(* Logix 5000 project; controller FRCFMS vendor 1 type 14 code 150 rev 33.11; software revision 33.00 *)
// FRCFMS

TASK MainTask (continuous, watchdog 500 ms) : MainProgram, ModbusSlaveTCP

MODULES
   Local : vendor 1 type 14 code 150 (Compact 0, rev 33.11)
      Counters : Embedded (Compact 3, rev 1.1, Output RPI 20 ms)
      Discrete_IO : Embedded (Compact 1, rev 3.1, Output RPI 20 ms)
      Analog_IO : Embedded (Compact 2, rev 1.1, Output RPI 80 ms)
      Blue_Driver_Station : vendor 1 type 7 code 357 (Ethernet 10.0.100.42, rev 1.1, Output RPI 20 ms)
      Red_Driver_Station : vendor 1 type 7 code 357 (Ethernet 10.0.100.41, rev 1.1, Output RPI 20 ms)
      Cargo_Ship : vendor 1 type 7 code 357 (Ethernet 10.0.100.43, rev 1.1, Output RPI 20 ms)
END_MODULES

TYPE AcceptResponse :
STRUCT
   Instance : DINT;
   Addr : SockAddr;
END_STRUCT
END_TYPE

TYPE READ_DATA_REQ :
STRUCT
   Timeout : DINT;
   BufLen : DINT;
END_STRUCT
END_TYPE

TYPE READ_RESP_STR :
STRUCT
   FromAddr : SockAddr;
   Buf : STR_4096;
END_STRUCT
END_TYPE

TYPE REQUEST_PARAMETERS :
STRUCT
   Type : DINT;
   Addr : SockAddr;
END_STRUCT
END_TYPE

TYPE SockAddr :
STRUCT
   Family : INT;
   Port : INT;
   Addr : DINT;
END_STRUCT
END_TYPE

TYPE STR_1 :
STRUCT
   LEN : DINT;
   DATA : SINT[1];
END_STRUCT
END_TYPE

TYPE STR_4096 :
STRUCT
   LEN : DINT;
   DATA : SINT[4096];
END_STRUCT
END_TYPE

TYPE STR_462 :
STRUCT
   LEN : DINT;
   DATA : SINT[462];
END_STRUCT
END_TYPE

TYPE STR_OUT :
STRUCT
   LEN : DINT;
   BUFF : SINT[480];
END_STRUCT
END_TYPE

TYPE WRT_DATA :
STRUCT
   Timeout : DINT;
   ToAddr : SockAddr;
   Buffer : STR_OUT;
END_STRUCT
END_TYPE

VAR_GLOBAL   (* controller tags *)
   AllianceDisconnectedFlasher : TIMER := (PRE := 1000, ACC := 928, EN := 1, TT := 1);
   BlueBypass1 : BOOL;
   BlueBypass2 : BOOL;
   BlueBypass3 : BOOL;
   BlueConnected1 : BOOL;
   BlueConnected2 : BOOL;
   BlueConnected3 : BOOL;
   BlueESTOP1 : ALIAS FOR Blue_Driver_Station:I.Data.1;
   BlueESTOP1Light : ALIAS FOR Blue_Driver_Station:O.Data.15;
   BlueESTOP2 : ALIAS FOR Blue_Driver_Station:I.Data.3;
   BlueESTOP2Light : ALIAS FOR Blue_Driver_Station:O.Data.13;
   BlueESTOP3 : ALIAS FOR Blue_Driver_Station:I.Data.5;
   BlueESTOP3Light : ALIAS FOR Blue_Driver_Station:O.Data.11;
   BlueSoftwareESTOP1 : BOOL;
   BlueSoftwareESTOP2 : BOOL;
   BlueSoftwareESTOP3 : BOOL;
   BlueStackStatus1 : ALIAS FOR Blue_Driver_Station:O.Data.14;
   BlueStackStatus2 : ALIAS FOR Blue_Driver_Station:O.Data.12;
   BlueStackStatus3 : ALIAS FOR Blue_Driver_Station:O.Data.10;
   EStop_Light_flasher : TIMER := (PRE := 750);
   Field_Reset_Green : BOOL;
   FieldESTOP : BOOL;
   FieldESTOPButton : ALIAS FOR Local:1:I.Data.0;
   FieldESTOPLight : ALIAS FOR Local:1:O.Data.0;
   Latch_reset : TIMER := (PRE := 50, ACC := 50, EN := 1, DN := 1);
   LostComm : TIMER := (PRE := 5000, ACC := 5000);
   MatchStart : BOOL;
   MatchStartONS : BOOL;
   MatchSYNC : TIMER := (PRE := 1000);
   MBTI_Buf_Len_Sent : DINT := 11;
   MBTI_Change_Log_MSG : MESSAGE;
        MessageParameters(ServiceCode := 16#0010, LocalElement := MBTU_Log_Enable, ...)
   MBTI_Conn_Acc_Timeout_MSG : MESSAGE;
        MessageParameters(ServiceCode := 16#0010, LocalElement := MBTU_Inactivity_Timeout, ...)
   MBTI_Conn_Accept_MSG : MESSAGE;
        MessageParameters(ServiceCode := 16#0050, LocalElement := MBTU_Sock_Accept_Timeout, DestinationTag := MBTI_Sock_Accept_Resp, ...)
   MBTI_ConnectionsLastErrors : DINT;
   MBTI_Create_Sock_MSG : MESSAGE;
        MessageParameters(ServiceCode := 16#004b, LocalElement := MBTI_Socket_Param, DestinationTag := MBTI_Instance, ...)
   MBTI_Delete_All_MSG : MESSAGE;
        MessageParameters(ServiceCode := 16#0051, ...)
   MBTI_Instance : DINT := 25408;
   MBTI_Read_Data_MSG_00 : MESSAGE;
        MessageParameters(ServiceCode := 16#004d, LocalElement := MBTI_Read_Data_Req[0], DestinationTag := MBTI_Read_Resp[0], ...)
   MBTI_Read_Data_MSG_01 : MESSAGE;
        MessageParameters(ServiceCode := 16#004d, LocalElement := MBTI_Read_Data_Req[0], DestinationTag := MBTI_Read_Resp[1], ...)
   MBTI_Read_Data_MSG_02 : MESSAGE;
        MessageParameters(ServiceCode := 16#004d, LocalElement := MBTI_Read_Data_Req[0], DestinationTag := MBTI_Read_Resp[2], ...)
   MBTI_Read_Data_MSG_03 : MESSAGE;
        MessageParameters(ServiceCode := 16#004d, LocalElement := MBTI_Read_Data_Req[0], DestinationTag := MBTI_Read_Resp[3], ...)
   MBTI_Read_Data_MSG_04 : MESSAGE;
        MessageParameters(ServiceCode := 16#004d, LocalElement := MBTI_Read_Data_Req[0], DestinationTag := MBTI_Read_Resp[4], ...)
   MBTI_Read_Data_MSG_05 : MESSAGE;
        MessageParameters(ServiceCode := 16#004d, LocalElement := MBTI_Read_Data_Req[0], DestinationTag := MBTI_Read_Resp[5], ...)
   MBTI_Read_Data_MSG_06 : MESSAGE;
        MessageParameters(ServiceCode := 16#004d, LocalElement := MBTI_Read_Data_Req[0], DestinationTag := MBTI_Read_Resp[6], ...)
   MBTI_Read_Data_MSG_07 : MESSAGE;
        MessageParameters(ServiceCode := 16#004d, LocalElement := MBTI_Read_Data_Req[0], DestinationTag := MBTI_Read_Resp[7], ...)
   MBTI_Read_Data_MSG_08 : MESSAGE;
        MessageParameters(ServiceCode := 16#004d, LocalElement := MBTI_Read_Data_Req[0], DestinationTag := MBTI_Read_Resp[8], ...)
   MBTI_Read_Data_MSG_09 : MESSAGE;
        MessageParameters(ServiceCode := 16#004d, LocalElement := MBTI_Read_Data_Req[0], DestinationTag := MBTI_Read_Resp[9], ...)
   MBTI_Read_Data_Req : READ_DATA_REQ[10] := ([0].BufLen := 484, [1].BufLen := 484, [2].BufLen := 484, [3].BufLen := 484, [4].BufLen := 484, [5].BufLen := 484, [6].BufLen := 484, [7].BufLen := 484, [8].BufLen := 484, [9].BufLen := 484);
   MBTI_Read_Done : BOOL[32];
   MBTI_Read_Resp : READ_RESP_STR[10] := ([3].Buf := '$04$FA$00$00$00$06$00$01$00$04$00$01');
   MBTI_RW_Inactivity : DINT := 3000;
   MBTI_RW_Inactivity_MSG : MESSAGE;
        MessageParameters(ServiceCode := 16#0010, LocalElement := MBTI_RW_Inactivity, ...)
   MBTI_Sock_Accept_Resp : AcceptResponse := (Instance := 32342, Addr.Family := 2, Addr.Port := -3789, Addr.Addr := 167797765);
   MBTI_Socket_Param : REQUEST_PARAMETERS := (Type := 1, Addr.Family := 2, Addr.Port := 502);
   MBTI_Total_Open : INT := 1;
   MBTI_Total_Open_MSG : MESSAGE;
        MessageParameters(ServiceCode := 16#000e, DestinationTag := MBTI_Total_Open, ...)
   MBTI_Write_Data_MSG_00 : MESSAGE;
        MessageParameters(ServiceCode := 16#004e, LocalElement := MBTI_Write_Data_Out[0], DestinationTag := MBTI_Buf_Len_Sent, ...)
   MBTI_Write_Data_MSG_01 : MESSAGE;
        MessageParameters(ServiceCode := 16#004e, LocalElement := MBTI_Write_Data_Out[1], DestinationTag := MBTI_Buf_Len_Sent, ...)
   MBTI_Write_Data_MSG_02 : MESSAGE;
        MessageParameters(ServiceCode := 16#004e, LocalElement := MBTI_Write_Data_Out[2], DestinationTag := MBTI_Buf_Len_Sent, ...)
   MBTI_Write_Data_MSG_03 : MESSAGE;
        MessageParameters(ServiceCode := 16#004e, LocalElement := MBTI_Write_Data_Out[3], DestinationTag := MBTI_Buf_Len_Sent, ...)
   MBTI_Write_Data_MSG_04 : MESSAGE;
        MessageParameters(ServiceCode := 16#004e, LocalElement := MBTI_Write_Data_Out[4], DestinationTag := MBTI_Buf_Len_Sent, ...)
   MBTI_Write_Data_MSG_05 : MESSAGE;
        MessageParameters(ServiceCode := 16#004e, LocalElement := MBTI_Write_Data_Out[5], DestinationTag := MBTI_Buf_Len_Sent, ...)
   MBTI_Write_Data_MSG_06 : MESSAGE;
        MessageParameters(ServiceCode := 16#004e, LocalElement := MBTI_Write_Data_Out[6], DestinationTag := MBTI_Buf_Len_Sent, ...)
   MBTI_Write_Data_MSG_07 : MESSAGE;
        MessageParameters(ServiceCode := 16#004e, LocalElement := MBTI_Write_Data_Out[7], DestinationTag := MBTI_Buf_Len_Sent, ...)
   MBTI_Write_Data_MSG_08 : MESSAGE;
        MessageParameters(ServiceCode := 16#004e, LocalElement := MBTI_Write_Data_Out[8], DestinationTag := MBTI_Buf_Len_Sent, ...)
   MBTI_Write_Data_MSG_09 : MESSAGE;
        MessageParameters(ServiceCode := 16#004e, LocalElement := MBTI_Write_Data_Out[9], DestinationTag := MBTI_Buf_Len_Sent, ...)
   MBTI_Write_Data_Out : WRT_DATA[10] := ([0].Timeout := 500, [0].ToAddr.Family := 2, [0].Buffer.LEN := 11, [0].Buffer.BUFF[1] := 113, [0].Buffer.BUFF[5] := 5, [0].Buffer.BUFF[6] := 1, [0].Buffer.BUFF[7] := 2, [0].Buffer.BUFF[8] := 2, [0].Buffer.BUFF[9] := 127, [0].Buffer.BUFF[22] := 25, [0].Buffer.BUFF[24] := 24, [0].Buffer.BUFF[26] := 25, [0].Buffer.BUFF[28] := 32, [0].Buffer.BUFF[30] := 125, [0].Buffer.BUFF[32] := 125, [0].Buffer.BUFF[57] := 39, [0].Buffer.BUFF[58] := 15, [0].Buffer.BUFF[130] := 60, [0].Buffer.BUFF[243] := 1, [0].Buffer.BUFF[244] := 77, [0].Buffer.BUFF[246] := -34, [0].Buffer.BUFF[248] := 119, [0].Buffer.BUFF[464] := -64, [0].Buffer.BUFF[465] := 47, [0].Buffer.BUFF[466] := 126, [0].Buffer.BUFF[467] := -15, [0].Buffer.BUFF[468] := 124, [0].Buffer.BUFF[471] := -128, [0].Buffer.BUFF[472] := 124, [0].Buffer.BUFF[475] := -128, [0].Buffer.BUFF[476] := -100, [0].Buffer.BUFF[477] := 75, [0].Buffer.BUFF[478] := 57, [0].Buffer.BUFF[479] := -15, [1].Timeout := 500, [1].Buffer.LEN := 12, [1].Buffer.BUFF[1] := 1, [1].Buffer.BUFF[5] := 6, [1].Buffer.BUFF[6] := 1, [1].Buffer.BUFF[7] := 15, [1].Buffer.BUFF[11] := 32, [1].Buffer.BUFF[22] := 25, [1].Buffer.BUFF[24] := 24, [1].Buffer.BUFF[26] := 25, [1].Buffer.BUFF[28] := 32, [1].Buffer.BUFF[30] := 125, [1].Buffer.BUFF[32] := 125, [1].Buffer.BUFF[57] := 39, [1].Buffer.BUFF[58] := 15, [1].Buffer.BUFF[130] := 60, [1].Buffer.BUFF[243] := 1, [1].Buffer.BUFF[244] := 77, [1].Buffer.BUFF[246] := -34, [1].Buffer.BUFF[248] := 119, [1].Buffer.BUFF[464] := -64, [1].Buffer.BUFF[465] := 47, [1].Buffer.BUFF[466] := 126, [1].Buffer.BUFF[467] := -15, [1].Buffer.BUFF[468] := 124, [1].Buffer.BUFF[471] := -128,
        [1].Buffer.BUFF[472] := 124, [1].Buffer.BUFF[475] := -128, [1].Buffer.BUFF[476] := -100, [1].Buffer.BUFF[477] := 75, [1].Buffer.BUFF[478] := 57, [1].Buffer.BUFF[479] := -15, [2].Timeout := 500, [2].Buffer.LEN := 12, [2].Buffer.BUFF[1] := 9, [2].Buffer.BUFF[5] := 6, [2].Buffer.BUFF[6] := 1, [2].Buffer.BUFF[7] := 15, [2].Buffer.BUFF[11] := 32, [2].Buffer.BUFF[22] := 25, [2].Buffer.BUFF[24] := 24, [2].Buffer.BUFF[26] := 25, [2].Buffer.BUFF[28] := 32, [2].Buffer.BUFF[30] := 125, [2].Buffer.BUFF[32] := 125, [2].Buffer.BUFF[57] := 39, [2].Buffer.BUFF[58] := 15, [2].Buffer.BUFF[130] := 60, [2].Buffer.BUFF[243] := 1, [2].Buffer.BUFF[244] := 77, [2].Buffer.BUFF[246] := -34, [2].Buffer.BUFF[248] := 119, [2].Buffer.BUFF[464] := -64, [2].Buffer.BUFF[465] := 47, [2].Buffer.BUFF[466] := 126, [2].Buffer.BUFF[467] := -15, [2].Buffer.BUFF[468] := 124, [2].Buffer.BUFF[471] := -128, [2].Buffer.BUFF[472] := 124, [2].Buffer.BUFF[475] := -128, [2].Buffer.BUFF[476] := -100, [2].Buffer.BUFF[477] := 75, [2].Buffer.BUFF[478] := 57, [2].Buffer.BUFF[479] := -15, [3].Timeout := 500, [3].Buffer.LEN := 12, [3].Buffer.BUFF[0] := 119, [3].Buffer.BUFF[1] := 87, [3].Buffer.BUFF[5] := 6, [3].Buffer.BUFF[6] := -1, [3].Buffer.BUFF[7] := 16, [3].Buffer.BUFF[9] := 59, [3].Buffer.BUFF[11] := 10, [3].Buffer.BUFF[12] := -34, [3].Buffer.BUFF[13] := 15, [3].Buffer.BUFF[14] := -1, [3].Buffer.BUFF[25] := 3, [3].Buffer.BUFF[26] := -25, [3].Buffer.BUFF[27] := 4, [3].Buffer.BUFF[28] := 68, [3].Buffer.BUFF[29] := 1, [3].Buffer.BUFF[30] := -68, [3].Buffer.BUFF[31] := 2, [3].Buffer.BUFF[32] := -102, [3].Buffer.BUFF[33] := 2, [3].Buffer.BUFF[34] := -104,
        [3].Buffer.BUFF[35] := 3, [3].Buffer.BUFF[36] := 9, [3].Buffer.BUFF[47] := 3, [3].Buffer.BUFF[48] := -25, [3].Buffer.BUFF[84] := 28, [3].Buffer.BUFF[87] := -128, [3].Buffer.BUFF[88] := 10, [3].Buffer.BUFF[91] := -128, [3].Buffer.BUFF[92] := 36, [3].Buffer.BUFF[93] := 36, [3].Buffer.BUFF[94] := 48, [3].Buffer.BUFF[95] := -15, [3].Buffer.BUFF[96] := -60, [3].Buffer.BUFF[97] := 16, [3].Buffer.BUFF[100] := 30, [3].Buffer.BUFF[101] := -119, [3].Buffer.BUFF[102] := 99, [3].Buffer.BUFF[103] := -36, [3].Buffer.BUFF[104] := 12, [3].Buffer.BUFF[108] := 1, [3].Buffer.BUFF[112] := 2, [3].Buffer.BUFF[114] := -10, [3].Buffer.BUFF[115] := 1, [3].Buffer.BUFF[124] := 10, [3].Buffer.BUFF[127] := -128, [3].Buffer.BUFF[128] := 8, [3].Buffer.BUFF[131] := -128, [3].Buffer.BUFF[132] := 36, [3].Buffer.BUFF[133] := 36, [3].Buffer.BUFF[134] := 48, [3].Buffer.BUFF[135] := -15, [3].Buffer.BUFF[136] := 52, [3].Buffer.BUFF[137] := 17, [3].Buffer.BUFF[140] := -61, [3].Buffer.BUFF[142] := 30, [3].Buffer.BUFF[143] := -38, [3].Buffer.BUFF[144] := 2, [3].Buffer.BUFF[148] := 33, [3].Buffer.BUFF[156] := 8, [3].Buffer.BUFF[159] := -128, [3].Buffer.BUFF[160] := 8, [3].Buffer.BUFF[163] := -128, [3].Buffer.BUFF[164] := 36, [3].Buffer.BUFF[165] := 36, [3].Buffer.BUFF[166] := 48, [3].Buffer.BUFF[167] := -15, [3].Buffer.BUFF[168] := 92, [3].Buffer.BUFF[169] := 17, [3].Buffer.BUFF[172] := -61, [3].Buffer.BUFF[174] := 113, [3].Buffer.BUFF[175] := -42, [3].Buffer.BUFF[176] := 2, [3].Buffer.BUFF[181] := 6, [3].Buffer.BUFF[188] := 8, [3].Buffer.BUFF[191] := -128, [3].Buffer.BUFF[192] := 28, [3].Buffer.BUFF[195] := -128, [3].Buffer.BUFF[196] := 36, [3].Buffer.BUFF[197] := 36, [3].Buffer.BUFF[198] := 48,
        [3].Buffer.BUFF[199] := -15, [3].Buffer.BUFF[200] := 124, [3].Buffer.BUFF[201] := 17, [3].Buffer.BUFF[204] := -50, [3].Buffer.BUFF[205] := -113, [3].Buffer.BUFF[206] := -83, [3].Buffer.BUFF[207] := -49, [3].Buffer.BUFF[208] := 88, [3].Buffer.BUFF[212] := 2, [3].Buffer.BUFF[216] := 4, [3].Buffer.BUFF[217] := 68, [3].Buffer.BUFF[300] := 28, [3].Buffer.BUFF[303] := -128, [3].Buffer.BUFF[304] := 8, [3].Buffer.BUFF[307] := -128, [3].Buffer.BUFF[308] := 36, [3].Buffer.BUFF[309] := 36, [3].Buffer.BUFF[310] := 48, [3].Buffer.BUFF[311] := -15, [3].Buffer.BUFF[312] := -100, [3].Buffer.BUFF[313] := 17, [3].Buffer.BUFF[316] := 104, [3].Buffer.BUFF[317] := -120, [3].Buffer.BUFF[318] := 86, [3].Buffer.BUFF[319] := -53, [3].Buffer.BUFF[320] := 8, [3].Buffer.BUFF[324] := 1, [3].Buffer.BUFF[328] := 3, [3].Buffer.BUFF[332] := 8, [3].Buffer.BUFF[335] := -128, [3].Buffer.BUFF[336] := 28, [3].Buffer.BUFF[337] := 80, [3].Buffer.BUFF[339] := -128, [3].Buffer.BUFF[340] := 36, [3].Buffer.BUFF[341] := 36, [3].Buffer.BUFF[342] := 48, [3].Buffer.BUFF[343] := -15, [3].Buffer.BUFF[344] := 12, [3].Buffer.BUFF[345] := 18, [3].Buffer.BUFF[348] := 75, [3].Buffer.BUFF[349] := -83, [3].Buffer.BUFF[350] := -121, [3].Buffer.BUFF[351] := -61, [3].Buffer.BUFF[352] := 4, [3].Buffer.BUFF[353] := 16, [3].Buffer.BUFF[356] := 20, [3].Buffer.BUFF[368] := -73, [3].Buffer.BUFF[369] := 83, [3].Buffer.BUFF[373] := 27, [3].Buffer.BUFF[374] := -1, [3].Buffer.BUFF[375] := 16, [3].Buffer.BUFF[377] := 59, [3].Buffer.BUFF[379] := 10, [3].Buffer.BUFF[380] := 20, [3].Buffer.BUFF[382] := 58, [3].Buffer.BUFF[401] := 18, [3].Buffer.BUFF[403] := 6, [3].Buffer.BUFF[404] := 125, [3].Buffer.BUFF[405] := 124, [3].Buffer.BUFF[409] := 6,
        [3].Buffer.BUFF[411] := 1, [3].Buffer.BUFF[413] := 18, [3].Buffer.BUFF[415] := 6, [3].Buffer.BUFF[416] := 125, [3].Buffer.BUFF[417] := 124, [3].Buffer.BUFF[421] := 6, [3].Buffer.BUFF[423] := 1, [3].Buffer.BUFF[425] := 18, [3].Buffer.BUFF[427] := 6, [3].Buffer.BUFF[428] := 125, [3].Buffer.BUFF[429] := 124, [3].Buffer.BUFF[433] := 6, [3].Buffer.BUFF[435] := 1, [3].Buffer.BUFF[437] := 18, [3].Buffer.BUFF[439] := 6, [3].Buffer.BUFF[440] := 125, [3].Buffer.BUFF[441] := 124, [3].Buffer.BUFF[445] := 6, [3].Buffer.BUFF[447] := 1, [3].Buffer.BUFF[449] := 18, [3].Buffer.BUFF[451] := 6, [3].Buffer.BUFF[452] := 125, [3].Buffer.BUFF[453] := 124, [3].Buffer.BUFF[457] := 6, [3].Buffer.BUFF[459] := 1, [3].Buffer.BUFF[461] := 18, [3].Buffer.BUFF[463] := 6, [3].Buffer.BUFF[464] := 125, [3].Buffer.BUFF[465] := 124, [3].Buffer.BUFF[469] := 6, [3].Buffer.BUFF[471] := 1, [3].Buffer.BUFF[473] := 18, [3].Buffer.BUFF[475] := 6, [3].Buffer.BUFF[476] := 125, [3].Buffer.BUFF[477] := 124, [4].Timeout := 500, [4].Buffer.LEN := 12, [4].Buffer.BUFF[0] := 119, [4].Buffer.BUFF[1] := 87, [4].Buffer.BUFF[5] := 6, [4].Buffer.BUFF[6] := -1, [4].Buffer.BUFF[7] := 16, [4].Buffer.BUFF[9] := 59, [4].Buffer.BUFF[11] := 10, [4].Buffer.BUFF[12] := -34, [4].Buffer.BUFF[13] := 15, [4].Buffer.BUFF[14] := -1, [4].Buffer.BUFF[25] := 3, [4].Buffer.BUFF[26] := -25, [4].Buffer.BUFF[27] := 4, [4].Buffer.BUFF[28] := 68, [4].Buffer.BUFF[29] := 1, [4].Buffer.BUFF[30] := -68, [4].Buffer.BUFF[31] := 2, [4].Buffer.BUFF[32] := -102, [4].Buffer.BUFF[33] := 2, [4].Buffer.BUFF[34] := -104, [4].Buffer.BUFF[35] := 3, [4].Buffer.BUFF[36] := 9, [4].Buffer.BUFF[47] := 3,
        [4].Buffer.BUFF[48] := -25, [4].Buffer.BUFF[84] := 28, [4].Buffer.BUFF[87] := -128, [4].Buffer.BUFF[88] := 10, [4].Buffer.BUFF[91] := -128, [4].Buffer.BUFF[92] := 36, [4].Buffer.BUFF[93] := 36, [4].Buffer.BUFF[94] := 48, [4].Buffer.BUFF[95] := -15, [4].Buffer.BUFF[96] := -60, [4].Buffer.BUFF[97] := 16, [4].Buffer.BUFF[100] := 30, [4].Buffer.BUFF[101] := -119, [4].Buffer.BUFF[102] := 99, [4].Buffer.BUFF[103] := -36, [4].Buffer.BUFF[104] := 12, [4].Buffer.BUFF[108] := 1, [4].Buffer.BUFF[112] := 2, [4].Buffer.BUFF[114] := -10, [4].Buffer.BUFF[115] := 1, [4].Buffer.BUFF[124] := 10, [4].Buffer.BUFF[127] := -128, [4].Buffer.BUFF[128] := 8, [4].Buffer.BUFF[131] := -128, [4].Buffer.BUFF[132] := 36, [4].Buffer.BUFF[133] := 36, [4].Buffer.BUFF[134] := 48, [4].Buffer.BUFF[135] := -15, [4].Buffer.BUFF[136] := 52, [4].Buffer.BUFF[137] := 17, [4].Buffer.BUFF[140] := -61, [4].Buffer.BUFF[142] := 30, [4].Buffer.BUFF[143] := -38, [4].Buffer.BUFF[144] := 2, [4].Buffer.BUFF[148] := 33, [4].Buffer.BUFF[156] := 8, [4].Buffer.BUFF[159] := -128, [4].Buffer.BUFF[160] := 8, [4].Buffer.BUFF[163] := -128, [4].Buffer.BUFF[164] := 36, [4].Buffer.BUFF[165] := 36, [4].Buffer.BUFF[166] := 48, [4].Buffer.BUFF[167] := -15, [4].Buffer.BUFF[168] := 92, [4].Buffer.BUFF[169] := 17, [4].Buffer.BUFF[172] := -61, [4].Buffer.BUFF[174] := 113, [4].Buffer.BUFF[175] := -42, [4].Buffer.BUFF[176] := 2, [4].Buffer.BUFF[181] := 6, [4].Buffer.BUFF[188] := 8, [4].Buffer.BUFF[191] := -128, [4].Buffer.BUFF[192] := 28, [4].Buffer.BUFF[195] := -128, [4].Buffer.BUFF[196] := 36, [4].Buffer.BUFF[197] := 36, [4].Buffer.BUFF[198] := 48, [4].Buffer.BUFF[199] := -15, [4].Buffer.BUFF[200] := 124, [4].Buffer.BUFF[201] := 17,
        [4].Buffer.BUFF[204] := -50, [4].Buffer.BUFF[205] := -113, [4].Buffer.BUFF[206] := -83, [4].Buffer.BUFF[207] := -49, [4].Buffer.BUFF[208] := 88, [4].Buffer.BUFF[212] := 2, [4].Buffer.BUFF[216] := 4, [4].Buffer.BUFF[217] := 68, [4].Buffer.BUFF[300] := 28, [4].Buffer.BUFF[303] := -128, [4].Buffer.BUFF[304] := 8, [4].Buffer.BUFF[307] := -128, [4].Buffer.BUFF[308] := 36, [4].Buffer.BUFF[309] := 36, [4].Buffer.BUFF[310] := 48, [4].Buffer.BUFF[311] := -15, [4].Buffer.BUFF[312] := -100, [4].Buffer.BUFF[313] := 17, [4].Buffer.BUFF[316] := 104, [4].Buffer.BUFF[317] := -120, [4].Buffer.BUFF[318] := 86, [4].Buffer.BUFF[319] := -53, [4].Buffer.BUFF[320] := 8, [4].Buffer.BUFF[324] := 1, [4].Buffer.BUFF[328] := 3, [4].Buffer.BUFF[332] := 8, [4].Buffer.BUFF[335] := -128, [4].Buffer.BUFF[336] := 28, [4].Buffer.BUFF[337] := 80, [4].Buffer.BUFF[339] := -128, [4].Buffer.BUFF[340] := 36, [4].Buffer.BUFF[341] := 36, [4].Buffer.BUFF[342] := 48, [4].Buffer.BUFF[343] := -15, [4].Buffer.BUFF[344] := 12, [4].Buffer.BUFF[345] := 18, [4].Buffer.BUFF[348] := 75, [4].Buffer.BUFF[349] := -83, [4].Buffer.BUFF[350] := -121, [4].Buffer.BUFF[351] := -61, [4].Buffer.BUFF[352] := 4, [4].Buffer.BUFF[353] := 16, [4].Buffer.BUFF[356] := 20, [4].Buffer.BUFF[368] := -73, [4].Buffer.BUFF[369] := 83, [4].Buffer.BUFF[373] := 27, [4].Buffer.BUFF[374] := -1, [4].Buffer.BUFF[375] := 16, [4].Buffer.BUFF[377] := 59, [4].Buffer.BUFF[379] := 10, [4].Buffer.BUFF[380] := 20, [4].Buffer.BUFF[382] := 58, [4].Buffer.BUFF[401] := 18, [4].Buffer.BUFF[403] := 6, [4].Buffer.BUFF[404] := 125, [4].Buffer.BUFF[405] := 124, [4].Buffer.BUFF[409] := 6, [4].Buffer.BUFF[411] := 1, [4].Buffer.BUFF[413] := 18, [4].Buffer.BUFF[415] := 6,
        [4].Buffer.BUFF[416] := 125, [4].Buffer.BUFF[417] := 124, [4].Buffer.BUFF[421] := 6, [4].Buffer.BUFF[423] := 1, [4].Buffer.BUFF[425] := 18, [4].Buffer.BUFF[427] := 6, [4].Buffer.BUFF[428] := 125, [4].Buffer.BUFF[429] := 124, [4].Buffer.BUFF[433] := 6, [4].Buffer.BUFF[435] := 1, [4].Buffer.BUFF[437] := 18, [4].Buffer.BUFF[439] := 6, [4].Buffer.BUFF[440] := 125, [4].Buffer.BUFF[441] := 124, [4].Buffer.BUFF[445] := 6, [4].Buffer.BUFF[447] := 1, [4].Buffer.BUFF[449] := 18, [4].Buffer.BUFF[451] := 6, [4].Buffer.BUFF[452] := 125, [4].Buffer.BUFF[453] := 124, [4].Buffer.BUFF[457] := 6, [4].Buffer.BUFF[459] := 1, [4].Buffer.BUFF[461] := 18, [4].Buffer.BUFF[463] := 6, [4].Buffer.BUFF[464] := 125, [4].Buffer.BUFF[465] := 124, [4].Buffer.BUFF[469] := 6, [4].Buffer.BUFF[471] := 1, [4].Buffer.BUFF[473] := 18, [4].Buffer.BUFF[475] := 6, [4].Buffer.BUFF[476] := 125, [4].Buffer.BUFF[477] := 124, [5].Timeout := 500, [5].Buffer.LEN := 12, [5].Buffer.BUFF[0] := 119, [5].Buffer.BUFF[1] := 87, [5].Buffer.BUFF[5] := 6, [5].Buffer.BUFF[6] := -1, [5].Buffer.BUFF[7] := 16, [5].Buffer.BUFF[9] := 59, [5].Buffer.BUFF[11] := 10, [5].Buffer.BUFF[12] := -34, [5].Buffer.BUFF[13] := 15, [5].Buffer.BUFF[14] := -1, [5].Buffer.BUFF[25] := 3, [5].Buffer.BUFF[26] := -25, [5].Buffer.BUFF[27] := 4, [5].Buffer.BUFF[28] := 68, [5].Buffer.BUFF[29] := 1, [5].Buffer.BUFF[30] := -68, [5].Buffer.BUFF[31] := 2, [5].Buffer.BUFF[32] := -102, [5].Buffer.BUFF[33] := 2, [5].Buffer.BUFF[34] := -104, [5].Buffer.BUFF[35] := 3, [5].Buffer.BUFF[36] := 9, [5].Buffer.BUFF[47] := 3, [5].Buffer.BUFF[48] := -25, [5].Buffer.BUFF[84] := 28, [5].Buffer.BUFF[87] := -128,
        [5].Buffer.BUFF[88] := 10, [5].Buffer.BUFF[91] := -128, [5].Buffer.BUFF[92] := 36, [5].Buffer.BUFF[93] := 36, [5].Buffer.BUFF[94] := 48, [5].Buffer.BUFF[95] := -15, [5].Buffer.BUFF[96] := -60, [5].Buffer.BUFF[97] := 16, [5].Buffer.BUFF[100] := 30, [5].Buffer.BUFF[101] := -119, [5].Buffer.BUFF[102] := 99, [5].Buffer.BUFF[103] := -36, [5].Buffer.BUFF[104] := 12, [5].Buffer.BUFF[108] := 1, [5].Buffer.BUFF[112] := 2, [5].Buffer.BUFF[114] := -10, [5].Buffer.BUFF[115] := 1, [5].Buffer.BUFF[124] := 10, [5].Buffer.BUFF[127] := -128, [5].Buffer.BUFF[128] := 8, [5].Buffer.BUFF[131] := -128, [5].Buffer.BUFF[132] := 36, [5].Buffer.BUFF[133] := 36, [5].Buffer.BUFF[134] := 48, [5].Buffer.BUFF[135] := -15, [5].Buffer.BUFF[136] := 52, [5].Buffer.BUFF[137] := 17, [5].Buffer.BUFF[140] := -61, [5].Buffer.BUFF[142] := 30, [5].Buffer.BUFF[143] := -38, [5].Buffer.BUFF[144] := 2, [5].Buffer.BUFF[148] := 33, [5].Buffer.BUFF[156] := 8, [5].Buffer.BUFF[159] := -128, [5].Buffer.BUFF[160] := 8, [5].Buffer.BUFF[163] := -128, [5].Buffer.BUFF[164] := 36, [5].Buffer.BUFF[165] := 36, [5].Buffer.BUFF[166] := 48, [5].Buffer.BUFF[167] := -15, [5].Buffer.BUFF[168] := 92, [5].Buffer.BUFF[169] := 17, [5].Buffer.BUFF[172] := -61, [5].Buffer.BUFF[174] := 113, [5].Buffer.BUFF[175] := -42, [5].Buffer.BUFF[176] := 2, [5].Buffer.BUFF[181] := 6, [5].Buffer.BUFF[188] := 8, [5].Buffer.BUFF[191] := -128, [5].Buffer.BUFF[192] := 28, [5].Buffer.BUFF[195] := -128, [5].Buffer.BUFF[196] := 36, [5].Buffer.BUFF[197] := 36, [5].Buffer.BUFF[198] := 48, [5].Buffer.BUFF[199] := -15, [5].Buffer.BUFF[200] := 124, [5].Buffer.BUFF[201] := 17, [5].Buffer.BUFF[204] := -50, [5].Buffer.BUFF[205] := -113, [5].Buffer.BUFF[206] := -83,
        [5].Buffer.BUFF[207] := -49, [5].Buffer.BUFF[208] := 88, [5].Buffer.BUFF[212] := 2, [5].Buffer.BUFF[216] := 4, [5].Buffer.BUFF[217] := 68, [5].Buffer.BUFF[300] := 28, [5].Buffer.BUFF[303] := -128, [5].Buffer.BUFF[304] := 8, [5].Buffer.BUFF[307] := -128, [5].Buffer.BUFF[308] := 36, [5].Buffer.BUFF[309] := 36, [5].Buffer.BUFF[310] := 48, [5].Buffer.BUFF[311] := -15, [5].Buffer.BUFF[312] := -100, [5].Buffer.BUFF[313] := 17, [5].Buffer.BUFF[316] := 104, [5].Buffer.BUFF[317] := -120, [5].Buffer.BUFF[318] := 86, [5].Buffer.BUFF[319] := -53, [5].Buffer.BUFF[320] := 8, [5].Buffer.BUFF[324] := 1, [5].Buffer.BUFF[328] := 3, [5].Buffer.BUFF[332] := 8, [5].Buffer.BUFF[335] := -128, [5].Buffer.BUFF[336] := 28, [5].Buffer.BUFF[337] := 80, [5].Buffer.BUFF[339] := -128, [5].Buffer.BUFF[340] := 36, [5].Buffer.BUFF[341] := 36, [5].Buffer.BUFF[342] := 48, [5].Buffer.BUFF[343] := -15, [5].Buffer.BUFF[344] := 12, [5].Buffer.BUFF[345] := 18, [5].Buffer.BUFF[348] := 75, [5].Buffer.BUFF[349] := -83, [5].Buffer.BUFF[350] := -121, [5].Buffer.BUFF[351] := -61, [5].Buffer.BUFF[352] := 4, [5].Buffer.BUFF[353] := 16, [5].Buffer.BUFF[356] := 20, [5].Buffer.BUFF[368] := -73, [5].Buffer.BUFF[369] := 83, [5].Buffer.BUFF[373] := 27, [5].Buffer.BUFF[374] := -1, [5].Buffer.BUFF[375] := 16, [5].Buffer.BUFF[377] := 59, [5].Buffer.BUFF[379] := 10, [5].Buffer.BUFF[380] := 20, [5].Buffer.BUFF[382] := 58, [5].Buffer.BUFF[401] := 18, [5].Buffer.BUFF[403] := 6, [5].Buffer.BUFF[404] := 125, [5].Buffer.BUFF[405] := 124, [5].Buffer.BUFF[409] := 6, [5].Buffer.BUFF[411] := 1, [5].Buffer.BUFF[413] := 18, [5].Buffer.BUFF[415] := 6, [5].Buffer.BUFF[416] := 125, [5].Buffer.BUFF[417] := 124, [5].Buffer.BUFF[421] := 6,
        [5].Buffer.BUFF[423] := 1, [5].Buffer.BUFF[425] := 18, [5].Buffer.BUFF[427] := 6, [5].Buffer.BUFF[428] := 125, [5].Buffer.BUFF[429] := 124, [5].Buffer.BUFF[433] := 6, [5].Buffer.BUFF[435] := 1, [5].Buffer.BUFF[437] := 18, [5].Buffer.BUFF[439] := 6, [5].Buffer.BUFF[440] := 125, [5].Buffer.BUFF[441] := 124, [5].Buffer.BUFF[445] := 6, [5].Buffer.BUFF[447] := 1, [5].Buffer.BUFF[449] := 18, [5].Buffer.BUFF[451] := 6, [5].Buffer.BUFF[452] := 125, [5].Buffer.BUFF[453] := 124, [5].Buffer.BUFF[457] := 6, [5].Buffer.BUFF[459] := 1, [5].Buffer.BUFF[461] := 18, [5].Buffer.BUFF[463] := 6, [5].Buffer.BUFF[464] := 125, [5].Buffer.BUFF[465] := 124, [5].Buffer.BUFF[469] := 6, [5].Buffer.BUFF[471] := 1, [5].Buffer.BUFF[473] := 18, [5].Buffer.BUFF[475] := 6, [5].Buffer.BUFF[476] := 125, [5].Buffer.BUFF[477] := 124, [6].Timeout := 500, [6].Buffer.LEN := 12, [6].Buffer.BUFF[0] := 119, [6].Buffer.BUFF[1] := 87, [6].Buffer.BUFF[5] := 6, [6].Buffer.BUFF[6] := -1, [6].Buffer.BUFF[7] := 16, [6].Buffer.BUFF[9] := 59, [6].Buffer.BUFF[11] := 10, [6].Buffer.BUFF[12] := -34, [6].Buffer.BUFF[13] := 15, [6].Buffer.BUFF[14] := -1, [6].Buffer.BUFF[25] := 3, [6].Buffer.BUFF[26] := -25, [6].Buffer.BUFF[27] := 4, [6].Buffer.BUFF[28] := 68, [6].Buffer.BUFF[29] := 1, [6].Buffer.BUFF[30] := -68, [6].Buffer.BUFF[31] := 2, [6].Buffer.BUFF[32] := -102, [6].Buffer.BUFF[33] := 2, [6].Buffer.BUFF[34] := -104, [6].Buffer.BUFF[35] := 3, [6].Buffer.BUFF[36] := 9, [6].Buffer.BUFF[47] := 3, [6].Buffer.BUFF[48] := -25, [6].Buffer.BUFF[84] := 28, [6].Buffer.BUFF[87] := -128, [6].Buffer.BUFF[88] := 10, [6].Buffer.BUFF[91] := -128, [6].Buffer.BUFF[92] := 36,
        [6].Buffer.BUFF[93] := 36, [6].Buffer.BUFF[94] := 48, [6].Buffer.BUFF[95] := -15, [6].Buffer.BUFF[96] := -60, [6].Buffer.BUFF[97] := 16, [6].Buffer.BUFF[100] := 30, [6].Buffer.BUFF[101] := -119, [6].Buffer.BUFF[102] := 99, [6].Buffer.BUFF[103] := -36, [6].Buffer.BUFF[104] := 12, [6].Buffer.BUFF[108] := 1, [6].Buffer.BUFF[112] := 2, [6].Buffer.BUFF[114] := -10, [6].Buffer.BUFF[115] := 1, [6].Buffer.BUFF[124] := 10, [6].Buffer.BUFF[127] := -128, [6].Buffer.BUFF[128] := 8, [6].Buffer.BUFF[131] := -128, [6].Buffer.BUFF[132] := 36, [6].Buffer.BUFF[133] := 36, [6].Buffer.BUFF[134] := 48, [6].Buffer.BUFF[135] := -15, [6].Buffer.BUFF[136] := 52, [6].Buffer.BUFF[137] := 17, [6].Buffer.BUFF[140] := -61, [6].Buffer.BUFF[142] := 30, [6].Buffer.BUFF[143] := -38, [6].Buffer.BUFF[144] := 2, [6].Buffer.BUFF[148] := 33, [6].Buffer.BUFF[156] := 8, [6].Buffer.BUFF[159] := -128, [6].Buffer.BUFF[160] := 8, [6].Buffer.BUFF[163] := -128, [6].Buffer.BUFF[164] := 36, [6].Buffer.BUFF[165] := 36, [6].Buffer.BUFF[166] := 48, [6].Buffer.BUFF[167] := -15, [6].Buffer.BUFF[168] := 92, [6].Buffer.BUFF[169] := 17, [6].Buffer.BUFF[172] := -61, [6].Buffer.BUFF[174] := 113, [6].Buffer.BUFF[175] := -42, [6].Buffer.BUFF[176] := 2, [6].Buffer.BUFF[181] := 6, [6].Buffer.BUFF[188] := 8, [6].Buffer.BUFF[191] := -128, [6].Buffer.BUFF[192] := 28, [6].Buffer.BUFF[195] := -128, [6].Buffer.BUFF[196] := 36, [6].Buffer.BUFF[197] := 36, [6].Buffer.BUFF[198] := 48, [6].Buffer.BUFF[199] := -15, [6].Buffer.BUFF[200] := 124, [6].Buffer.BUFF[201] := 17, [6].Buffer.BUFF[204] := -50, [6].Buffer.BUFF[205] := -113, [6].Buffer.BUFF[206] := -83, [6].Buffer.BUFF[207] := -49, [6].Buffer.BUFF[208] := 88, [6].Buffer.BUFF[212] := 2,
        [6].Buffer.BUFF[216] := 4, [6].Buffer.BUFF[217] := 68, [6].Buffer.BUFF[300] := 28, [6].Buffer.BUFF[303] := -128, [6].Buffer.BUFF[304] := 8, [6].Buffer.BUFF[307] := -128, [6].Buffer.BUFF[308] := 36, [6].Buffer.BUFF[309] := 36, [6].Buffer.BUFF[310] := 48, [6].Buffer.BUFF[311] := -15, [6].Buffer.BUFF[312] := -100, [6].Buffer.BUFF[313] := 17, [6].Buffer.BUFF[316] := 104, [6].Buffer.BUFF[317] := -120, [6].Buffer.BUFF[318] := 86, [6].Buffer.BUFF[319] := -53, [6].Buffer.BUFF[320] := 8, [6].Buffer.BUFF[324] := 1, [6].Buffer.BUFF[328] := 3, [6].Buffer.BUFF[332] := 8, [6].Buffer.BUFF[335] := -128, [6].Buffer.BUFF[336] := 28, [6].Buffer.BUFF[337] := 80, [6].Buffer.BUFF[339] := -128, [6].Buffer.BUFF[340] := 36, [6].Buffer.BUFF[341] := 36, [6].Buffer.BUFF[342] := 48, [6].Buffer.BUFF[343] := -15, [6].Buffer.BUFF[344] := 12, [6].Buffer.BUFF[345] := 18, [6].Buffer.BUFF[348] := 75, [6].Buffer.BUFF[349] := -83, [6].Buffer.BUFF[350] := -121, [6].Buffer.BUFF[351] := -61, [6].Buffer.BUFF[352] := 4, [6].Buffer.BUFF[353] := 16, [6].Buffer.BUFF[356] := 20, [6].Buffer.BUFF[368] := -73, [6].Buffer.BUFF[369] := 83, [6].Buffer.BUFF[373] := 27, [6].Buffer.BUFF[374] := -1, [6].Buffer.BUFF[375] := 16, [6].Buffer.BUFF[377] := 59, [6].Buffer.BUFF[379] := 10, [6].Buffer.BUFF[380] := 20, [6].Buffer.BUFF[382] := 58, [6].Buffer.BUFF[401] := 18, [6].Buffer.BUFF[403] := 6, [6].Buffer.BUFF[404] := 125, [6].Buffer.BUFF[405] := 124, [6].Buffer.BUFF[409] := 6, [6].Buffer.BUFF[411] := 1, [6].Buffer.BUFF[413] := 18, [6].Buffer.BUFF[415] := 6, [6].Buffer.BUFF[416] := 125, [6].Buffer.BUFF[417] := 124, [6].Buffer.BUFF[421] := 6, [6].Buffer.BUFF[423] := 1, [6].Buffer.BUFF[425] := 18, [6].Buffer.BUFF[427] := 6,
        [6].Buffer.BUFF[428] := 125, [6].Buffer.BUFF[429] := 124, [6].Buffer.BUFF[433] := 6, [6].Buffer.BUFF[435] := 1, [6].Buffer.BUFF[437] := 18, [6].Buffer.BUFF[439] := 6, [6].Buffer.BUFF[440] := 125, [6].Buffer.BUFF[441] := 124, [6].Buffer.BUFF[445] := 6, [6].Buffer.BUFF[447] := 1, [6].Buffer.BUFF[449] := 18, [6].Buffer.BUFF[451] := 6, [6].Buffer.BUFF[452] := 125, [6].Buffer.BUFF[453] := 124, [6].Buffer.BUFF[457] := 6, [6].Buffer.BUFF[459] := 1, [6].Buffer.BUFF[461] := 18, [6].Buffer.BUFF[463] := 6, [6].Buffer.BUFF[464] := 125, [6].Buffer.BUFF[465] := 124, [6].Buffer.BUFF[469] := 6, [6].Buffer.BUFF[471] := 1, [6].Buffer.BUFF[473] := 18, [6].Buffer.BUFF[475] := 6, [6].Buffer.BUFF[476] := 125, [6].Buffer.BUFF[477] := 124, [7].Timeout := 500, [7].Buffer.LEN := 12, [7].Buffer.BUFF[0] := 119, [7].Buffer.BUFF[1] := 87, [7].Buffer.BUFF[5] := 6, [7].Buffer.BUFF[6] := -1, [7].Buffer.BUFF[7] := 16, [7].Buffer.BUFF[9] := 59, [7].Buffer.BUFF[11] := 10, [7].Buffer.BUFF[12] := -34, [7].Buffer.BUFF[13] := 15, [7].Buffer.BUFF[14] := -1, [7].Buffer.BUFF[25] := 3, [7].Buffer.BUFF[26] := -25, [7].Buffer.BUFF[27] := 4, [7].Buffer.BUFF[28] := 68, [7].Buffer.BUFF[29] := 1, [7].Buffer.BUFF[30] := -68, [7].Buffer.BUFF[31] := 2, [7].Buffer.BUFF[32] := -102, [7].Buffer.BUFF[33] := 2, [7].Buffer.BUFF[34] := -104, [7].Buffer.BUFF[35] := 3, [7].Buffer.BUFF[36] := 9, [7].Buffer.BUFF[47] := 3, [7].Buffer.BUFF[48] := -25, [7].Buffer.BUFF[84] := 28, [7].Buffer.BUFF[87] := -128, [7].Buffer.BUFF[88] := 10, [7].Buffer.BUFF[91] := -128, [7].Buffer.BUFF[92] := 36, [7].Buffer.BUFF[93] := 36, [7].Buffer.BUFF[94] := 48, [7].Buffer.BUFF[95] := -15,
        [7].Buffer.BUFF[96] := -60, [7].Buffer.BUFF[97] := 16, [7].Buffer.BUFF[100] := 30, [7].Buffer.BUFF[101] := -119, [7].Buffer.BUFF[102] := 99, [7].Buffer.BUFF[103] := -36, [7].Buffer.BUFF[104] := 12, [7].Buffer.BUFF[108] := 1, [7].Buffer.BUFF[112] := 2, [7].Buffer.BUFF[114] := -10, [7].Buffer.BUFF[115] := 1, [7].Buffer.BUFF[124] := 10, [7].Buffer.BUFF[127] := -128, [7].Buffer.BUFF[128] := 8, [7].Buffer.BUFF[131] := -128, [7].Buffer.BUFF[132] := 36, [7].Buffer.BUFF[133] := 36, [7].Buffer.BUFF[134] := 48, [7].Buffer.BUFF[135] := -15, [7].Buffer.BUFF[136] := 52, [7].Buffer.BUFF[137] := 17, [7].Buffer.BUFF[140] := -61, [7].Buffer.BUFF[142] := 30, [7].Buffer.BUFF[143] := -38, [7].Buffer.BUFF[144] := 2, [7].Buffer.BUFF[148] := 33, [7].Buffer.BUFF[156] := 8, [7].Buffer.BUFF[159] := -128, [7].Buffer.BUFF[160] := 8, [7].Buffer.BUFF[163] := -128, [7].Buffer.BUFF[164] := 36, [7].Buffer.BUFF[165] := 36, [7].Buffer.BUFF[166] := 48, [7].Buffer.BUFF[167] := -15, [7].Buffer.BUFF[168] := 92, [7].Buffer.BUFF[169] := 17, [7].Buffer.BUFF[172] := -61, [7].Buffer.BUFF[174] := 113, [7].Buffer.BUFF[175] := -42, [7].Buffer.BUFF[176] := 2, [7].Buffer.BUFF[181] := 6, [7].Buffer.BUFF[188] := 8, [7].Buffer.BUFF[191] := -128, [7].Buffer.BUFF[192] := 28, [7].Buffer.BUFF[195] := -128, [7].Buffer.BUFF[196] := 36, [7].Buffer.BUFF[197] := 36, [7].Buffer.BUFF[198] := 48, [7].Buffer.BUFF[199] := -15, [7].Buffer.BUFF[200] := 124, [7].Buffer.BUFF[201] := 17, [7].Buffer.BUFF[204] := -50, [7].Buffer.BUFF[205] := -113, [7].Buffer.BUFF[206] := -83, [7].Buffer.BUFF[207] := -49, [7].Buffer.BUFF[208] := 88, [7].Buffer.BUFF[212] := 2, [7].Buffer.BUFF[216] := 4, [7].Buffer.BUFF[217] := 68, [7].Buffer.BUFF[300] := 28,
        [7].Buffer.BUFF[303] := -128, [7].Buffer.BUFF[304] := 8, [7].Buffer.BUFF[307] := -128, [7].Buffer.BUFF[308] := 36, [7].Buffer.BUFF[309] := 36, [7].Buffer.BUFF[310] := 48, [7].Buffer.BUFF[311] := -15, [7].Buffer.BUFF[312] := -100, [7].Buffer.BUFF[313] := 17, [7].Buffer.BUFF[316] := 104, [7].Buffer.BUFF[317] := -120, [7].Buffer.BUFF[318] := 86, [7].Buffer.BUFF[319] := -53, [7].Buffer.BUFF[320] := 8, [7].Buffer.BUFF[324] := 1, [7].Buffer.BUFF[328] := 3, [7].Buffer.BUFF[332] := 8, [7].Buffer.BUFF[335] := -128, [7].Buffer.BUFF[336] := 28, [7].Buffer.BUFF[337] := 80, [7].Buffer.BUFF[339] := -128, [7].Buffer.BUFF[340] := 36, [7].Buffer.BUFF[341] := 36, [7].Buffer.BUFF[342] := 48, [7].Buffer.BUFF[343] := -15, [7].Buffer.BUFF[344] := 12, [7].Buffer.BUFF[345] := 18, [7].Buffer.BUFF[348] := 75, [7].Buffer.BUFF[349] := -83, [7].Buffer.BUFF[350] := -121, [7].Buffer.BUFF[351] := -61, [7].Buffer.BUFF[352] := 4, [7].Buffer.BUFF[353] := 16, [7].Buffer.BUFF[356] := 20, [7].Buffer.BUFF[368] := -73, [7].Buffer.BUFF[369] := 83, [7].Buffer.BUFF[373] := 27, [7].Buffer.BUFF[374] := -1, [7].Buffer.BUFF[375] := 16, [7].Buffer.BUFF[377] := 59, [7].Buffer.BUFF[379] := 10, [7].Buffer.BUFF[380] := 20, [7].Buffer.BUFF[382] := 58, [7].Buffer.BUFF[401] := 18, [7].Buffer.BUFF[403] := 6, [7].Buffer.BUFF[404] := 125, [7].Buffer.BUFF[405] := 124, [7].Buffer.BUFF[409] := 6, [7].Buffer.BUFF[411] := 1, [7].Buffer.BUFF[413] := 18, [7].Buffer.BUFF[415] := 6, [7].Buffer.BUFF[416] := 125, [7].Buffer.BUFF[417] := 124, [7].Buffer.BUFF[421] := 6, [7].Buffer.BUFF[423] := 1, [7].Buffer.BUFF[425] := 18, [7].Buffer.BUFF[427] := 6, [7].Buffer.BUFF[428] := 125, [7].Buffer.BUFF[429] := 124, [7].Buffer.BUFF[433] := 6,
        [7].Buffer.BUFF[435] := 1, [7].Buffer.BUFF[437] := 18, [7].Buffer.BUFF[439] := 6, [7].Buffer.BUFF[440] := 125, [7].Buffer.BUFF[441] := 124, [7].Buffer.BUFF[445] := 6, [7].Buffer.BUFF[447] := 1, [7].Buffer.BUFF[449] := 18, [7].Buffer.BUFF[451] := 6, [7].Buffer.BUFF[452] := 125, [7].Buffer.BUFF[453] := 124, [7].Buffer.BUFF[457] := 6, [7].Buffer.BUFF[459] := 1, [7].Buffer.BUFF[461] := 18, [7].Buffer.BUFF[463] := 6, [7].Buffer.BUFF[464] := 125, [7].Buffer.BUFF[465] := 124, [7].Buffer.BUFF[469] := 6, [7].Buffer.BUFF[471] := 1, [7].Buffer.BUFF[473] := 18, [7].Buffer.BUFF[475] := 6, [7].Buffer.BUFF[476] := 125, [7].Buffer.BUFF[477] := 124, [8].Timeout := 500, [8].Buffer.LEN := 12, [8].Buffer.BUFF[0] := 119, [8].Buffer.BUFF[1] := 87, [8].Buffer.BUFF[5] := 6, [8].Buffer.BUFF[6] := -1, [8].Buffer.BUFF[7] := 16, [8].Buffer.BUFF[9] := 59, [8].Buffer.BUFF[11] := 10, [8].Buffer.BUFF[12] := -34, [8].Buffer.BUFF[13] := 15, [8].Buffer.BUFF[14] := -1, [8].Buffer.BUFF[25] := 3, [8].Buffer.BUFF[26] := -25, [8].Buffer.BUFF[27] := 4, [8].Buffer.BUFF[28] := 68, [8].Buffer.BUFF[29] := 1, [8].Buffer.BUFF[30] := -68, [8].Buffer.BUFF[31] := 2, [8].Buffer.BUFF[32] := -102, [8].Buffer.BUFF[33] := 2, [8].Buffer.BUFF[34] := -104, [8].Buffer.BUFF[35] := 3, [8].Buffer.BUFF[36] := 9, [8].Buffer.BUFF[47] := 3, [8].Buffer.BUFF[48] := -25, [8].Buffer.BUFF[84] := 28, [8].Buffer.BUFF[87] := -128, [8].Buffer.BUFF[88] := 10, [8].Buffer.BUFF[91] := -128, [8].Buffer.BUFF[92] := 36, [8].Buffer.BUFF[93] := 36, [8].Buffer.BUFF[94] := 48, [8].Buffer.BUFF[95] := -15, [8].Buffer.BUFF[96] := -60, [8].Buffer.BUFF[97] := 16, [8].Buffer.BUFF[100] := 30,
        [8].Buffer.BUFF[101] := -119, [8].Buffer.BUFF[102] := 99, [8].Buffer.BUFF[103] := -36, [8].Buffer.BUFF[104] := 12, [8].Buffer.BUFF[108] := 1, [8].Buffer.BUFF[112] := 2, [8].Buffer.BUFF[114] := -10, [8].Buffer.BUFF[115] := 1, [8].Buffer.BUFF[124] := 10, [8].Buffer.BUFF[127] := -128, [8].Buffer.BUFF[128] := 8, [8].Buffer.BUFF[131] := -128, [8].Buffer.BUFF[132] := 36, [8].Buffer.BUFF[133] := 36, [8].Buffer.BUFF[134] := 48, [8].Buffer.BUFF[135] := -15, [8].Buffer.BUFF[136] := 52, [8].Buffer.BUFF[137] := 17, [8].Buffer.BUFF[140] := -61, [8].Buffer.BUFF[142] := 30, [8].Buffer.BUFF[143] := -38, [8].Buffer.BUFF[144] := 2, [8].Buffer.BUFF[148] := 33, [8].Buffer.BUFF[156] := 8, [8].Buffer.BUFF[159] := -128, [8].Buffer.BUFF[160] := 8, [8].Buffer.BUFF[163] := -128, [8].Buffer.BUFF[164] := 36, [8].Buffer.BUFF[165] := 36, [8].Buffer.BUFF[166] := 48, [8].Buffer.BUFF[167] := -15, [8].Buffer.BUFF[168] := 92, [8].Buffer.BUFF[169] := 17, [8].Buffer.BUFF[172] := -61, [8].Buffer.BUFF[174] := 113, [8].Buffer.BUFF[175] := -42, [8].Buffer.BUFF[176] := 2, [8].Buffer.BUFF[181] := 6, [8].Buffer.BUFF[188] := 8, [8].Buffer.BUFF[191] := -128, [8].Buffer.BUFF[192] := 28, [8].Buffer.BUFF[195] := -128, [8].Buffer.BUFF[196] := 36, [8].Buffer.BUFF[197] := 36, [8].Buffer.BUFF[198] := 48, [8].Buffer.BUFF[199] := -15, [8].Buffer.BUFF[200] := 124, [8].Buffer.BUFF[201] := 17, [8].Buffer.BUFF[204] := -50, [8].Buffer.BUFF[205] := -113, [8].Buffer.BUFF[206] := -83, [8].Buffer.BUFF[207] := -49, [8].Buffer.BUFF[208] := 88, [8].Buffer.BUFF[212] := 2, [8].Buffer.BUFF[216] := 4, [8].Buffer.BUFF[217] := 68, [8].Buffer.BUFF[300] := 28, [8].Buffer.BUFF[303] := -128, [8].Buffer.BUFF[304] := 8, [8].Buffer.BUFF[307] := -128,
        [8].Buffer.BUFF[308] := 36, [8].Buffer.BUFF[309] := 36, [8].Buffer.BUFF[310] := 48, [8].Buffer.BUFF[311] := -15, [8].Buffer.BUFF[312] := -100, [8].Buffer.BUFF[313] := 17, [8].Buffer.BUFF[316] := 104, [8].Buffer.BUFF[317] := -120, [8].Buffer.BUFF[318] := 86, [8].Buffer.BUFF[319] := -53, [8].Buffer.BUFF[320] := 8, [8].Buffer.BUFF[324] := 1, [8].Buffer.BUFF[328] := 3, [8].Buffer.BUFF[332] := 8, [8].Buffer.BUFF[335] := -128, [8].Buffer.BUFF[336] := 28, [8].Buffer.BUFF[337] := 80, [8].Buffer.BUFF[339] := -128, [8].Buffer.BUFF[340] := 36, [8].Buffer.BUFF[341] := 36, [8].Buffer.BUFF[342] := 48, [8].Buffer.BUFF[343] := -15, [8].Buffer.BUFF[344] := 12, [8].Buffer.BUFF[345] := 18, [8].Buffer.BUFF[348] := 75, [8].Buffer.BUFF[349] := -83, [8].Buffer.BUFF[350] := -121, [8].Buffer.BUFF[351] := -61, [8].Buffer.BUFF[352] := 4, [8].Buffer.BUFF[353] := 16, [8].Buffer.BUFF[356] := 20, [8].Buffer.BUFF[368] := -73, [8].Buffer.BUFF[369] := 83, [8].Buffer.BUFF[373] := 27, [8].Buffer.BUFF[374] := -1, [8].Buffer.BUFF[375] := 16, [8].Buffer.BUFF[377] := 59, [8].Buffer.BUFF[379] := 10, [8].Buffer.BUFF[380] := 20, [8].Buffer.BUFF[382] := 58, [8].Buffer.BUFF[401] := 18, [8].Buffer.BUFF[403] := 6, [8].Buffer.BUFF[404] := 125, [8].Buffer.BUFF[405] := 124, [8].Buffer.BUFF[409] := 6, [8].Buffer.BUFF[411] := 1, [8].Buffer.BUFF[413] := 18, [8].Buffer.BUFF[415] := 6, [8].Buffer.BUFF[416] := 125, [8].Buffer.BUFF[417] := 124, [8].Buffer.BUFF[421] := 6, [8].Buffer.BUFF[423] := 1, [8].Buffer.BUFF[425] := 18, [8].Buffer.BUFF[427] := 6, [8].Buffer.BUFF[428] := 125, [8].Buffer.BUFF[429] := 124, [8].Buffer.BUFF[433] := 6, [8].Buffer.BUFF[435] := 1, [8].Buffer.BUFF[437] := 18, [8].Buffer.BUFF[439] := 6,
        [8].Buffer.BUFF[440] := 125, [8].Buffer.BUFF[441] := 124, [8].Buffer.BUFF[445] := 6, [8].Buffer.BUFF[447] := 1, [8].Buffer.BUFF[449] := 18, [8].Buffer.BUFF[451] := 6, [8].Buffer.BUFF[452] := 125, [8].Buffer.BUFF[453] := 124, [8].Buffer.BUFF[457] := 6, [8].Buffer.BUFF[459] := 1, [8].Buffer.BUFF[461] := 18, [8].Buffer.BUFF[463] := 6, [8].Buffer.BUFF[464] := 125, [8].Buffer.BUFF[465] := 124, [8].Buffer.BUFF[469] := 6, [8].Buffer.BUFF[471] := 1, [8].Buffer.BUFF[473] := 18, [8].Buffer.BUFF[475] := 6, [8].Buffer.BUFF[476] := 125, [8].Buffer.BUFF[477] := 124, [9].Timeout := 500, [9].Buffer.LEN := 12, [9].Buffer.BUFF[0] := 119, [9].Buffer.BUFF[1] := 87, [9].Buffer.BUFF[5] := 6, [9].Buffer.BUFF[6] := -1, [9].Buffer.BUFF[7] := 16, [9].Buffer.BUFF[9] := 59, [9].Buffer.BUFF[11] := 10, [9].Buffer.BUFF[12] := -34, [9].Buffer.BUFF[13] := 15, [9].Buffer.BUFF[14] := -1, [9].Buffer.BUFF[25] := 3, [9].Buffer.BUFF[26] := -25, [9].Buffer.BUFF[27] := 4, [9].Buffer.BUFF[28] := 68, [9].Buffer.BUFF[29] := 1, [9].Buffer.BUFF[30] := -68, [9].Buffer.BUFF[31] := 2, [9].Buffer.BUFF[32] := -102, [9].Buffer.BUFF[33] := 2, [9].Buffer.BUFF[34] := -104, [9].Buffer.BUFF[35] := 3, [9].Buffer.BUFF[36] := 9, [9].Buffer.BUFF[47] := 3, [9].Buffer.BUFF[48] := -25, [9].Buffer.BUFF[84] := 28, [9].Buffer.BUFF[87] := -128, [9].Buffer.BUFF[88] := 10, [9].Buffer.BUFF[91] := -128, [9].Buffer.BUFF[92] := 36, [9].Buffer.BUFF[93] := 36, [9].Buffer.BUFF[94] := 48, [9].Buffer.BUFF[95] := -15, [9].Buffer.BUFF[96] := -60, [9].Buffer.BUFF[97] := 16, [9].Buffer.BUFF[100] := 30, [9].Buffer.BUFF[101] := -119, [9].Buffer.BUFF[102] := 99, [9].Buffer.BUFF[103] := -36,
        [9].Buffer.BUFF[104] := 12, [9].Buffer.BUFF[108] := 1, [9].Buffer.BUFF[112] := 2, [9].Buffer.BUFF[114] := -10, [9].Buffer.BUFF[115] := 1, [9].Buffer.BUFF[124] := 10, [9].Buffer.BUFF[127] := -128, [9].Buffer.BUFF[128] := 8, [9].Buffer.BUFF[131] := -128, [9].Buffer.BUFF[132] := 36, [9].Buffer.BUFF[133] := 36, [9].Buffer.BUFF[134] := 48, [9].Buffer.BUFF[135] := -15, [9].Buffer.BUFF[136] := 52, [9].Buffer.BUFF[137] := 17, [9].Buffer.BUFF[140] := -61, [9].Buffer.BUFF[142] := 30, [9].Buffer.BUFF[143] := -38, [9].Buffer.BUFF[144] := 2, [9].Buffer.BUFF[148] := 33, [9].Buffer.BUFF[156] := 8, [9].Buffer.BUFF[159] := -128, [9].Buffer.BUFF[160] := 8, [9].Buffer.BUFF[163] := -128, [9].Buffer.BUFF[164] := 36, [9].Buffer.BUFF[165] := 36, [9].Buffer.BUFF[166] := 48, [9].Buffer.BUFF[167] := -15, [9].Buffer.BUFF[168] := 92, [9].Buffer.BUFF[169] := 17, [9].Buffer.BUFF[172] := -61, [9].Buffer.BUFF[174] := 113, [9].Buffer.BUFF[175] := -42, [9].Buffer.BUFF[176] := 2, [9].Buffer.BUFF[181] := 6, [9].Buffer.BUFF[188] := 8, [9].Buffer.BUFF[191] := -128, [9].Buffer.BUFF[192] := 28, [9].Buffer.BUFF[195] := -128, [9].Buffer.BUFF[196] := 36, [9].Buffer.BUFF[197] := 36, [9].Buffer.BUFF[198] := 48, [9].Buffer.BUFF[199] := -15, [9].Buffer.BUFF[200] := 124, [9].Buffer.BUFF[201] := 17, [9].Buffer.BUFF[204] := -50, [9].Buffer.BUFF[205] := -113, [9].Buffer.BUFF[206] := -83, [9].Buffer.BUFF[207] := -49, [9].Buffer.BUFF[208] := 88, [9].Buffer.BUFF[212] := 2, [9].Buffer.BUFF[216] := 4, [9].Buffer.BUFF[217] := 68, [9].Buffer.BUFF[300] := 28, [9].Buffer.BUFF[303] := -128, [9].Buffer.BUFF[304] := 8, [9].Buffer.BUFF[307] := -128, [9].Buffer.BUFF[308] := 36, [9].Buffer.BUFF[309] := 36, [9].Buffer.BUFF[310] := 48,
        [9].Buffer.BUFF[311] := -15, [9].Buffer.BUFF[312] := -100, [9].Buffer.BUFF[313] := 17, [9].Buffer.BUFF[316] := 104, [9].Buffer.BUFF[317] := -120, [9].Buffer.BUFF[318] := 86, [9].Buffer.BUFF[319] := -53, [9].Buffer.BUFF[320] := 8, [9].Buffer.BUFF[324] := 1, [9].Buffer.BUFF[328] := 3, [9].Buffer.BUFF[332] := 8, [9].Buffer.BUFF[335] := -128, [9].Buffer.BUFF[336] := 28, [9].Buffer.BUFF[337] := 80, [9].Buffer.BUFF[339] := -128, [9].Buffer.BUFF[340] := 36, [9].Buffer.BUFF[341] := 36, [9].Buffer.BUFF[342] := 48, [9].Buffer.BUFF[343] := -15, [9].Buffer.BUFF[344] := 12, [9].Buffer.BUFF[345] := 18, [9].Buffer.BUFF[348] := 75, [9].Buffer.BUFF[349] := -83, [9].Buffer.BUFF[350] := -121, [9].Buffer.BUFF[351] := -61, [9].Buffer.BUFF[352] := 4, [9].Buffer.BUFF[353] := 16, [9].Buffer.BUFF[356] := 20, [9].Buffer.BUFF[368] := -73, [9].Buffer.BUFF[369] := 83, [9].Buffer.BUFF[373] := 27, [9].Buffer.BUFF[374] := -1, [9].Buffer.BUFF[375] := 16, [9].Buffer.BUFF[377] := 59, [9].Buffer.BUFF[379] := 10, [9].Buffer.BUFF[380] := 20, [9].Buffer.BUFF[382] := 58, [9].Buffer.BUFF[401] := 18, [9].Buffer.BUFF[403] := 6, [9].Buffer.BUFF[404] := 125, [9].Buffer.BUFF[405] := 124, [9].Buffer.BUFF[409] := 6, [9].Buffer.BUFF[411] := 1, [9].Buffer.BUFF[413] := 18, [9].Buffer.BUFF[415] := 6, [9].Buffer.BUFF[416] := 125, [9].Buffer.BUFF[417] := 124, [9].Buffer.BUFF[421] := 6, [9].Buffer.BUFF[423] := 1, [9].Buffer.BUFF[425] := 18, [9].Buffer.BUFF[427] := 6, [9].Buffer.BUFF[428] := 125, [9].Buffer.BUFF[429] := 124, [9].Buffer.BUFF[433] := 6, [9].Buffer.BUFF[435] := 1, [9].Buffer.BUFF[437] := 18, [9].Buffer.BUFF[439] := 6, [9].Buffer.BUFF[440] := 125, [9].Buffer.BUFF[441] := 124, [9].Buffer.BUFF[445] := 6,
        [9].Buffer.BUFF[447] := 1, [9].Buffer.BUFF[449] := 18, [9].Buffer.BUFF[451] := 6, [9].Buffer.BUFF[452] := 125, [9].Buffer.BUFF[453] := 124, [9].Buffer.BUFF[457] := 6, [9].Buffer.BUFF[459] := 1, [9].Buffer.BUFF[461] := 18, [9].Buffer.BUFF[463] := 6, [9].Buffer.BUFF[464] := 125, [9].Buffer.BUFF[465] := 124, [9].Buffer.BUFF[469] := 6, [9].Buffer.BUFF[471] := 1, [9].Buffer.BUFF[473] := 18, [9].Buffer.BUFF[475] := 6, [9].Buffer.BUFF[476] := 125, [9].Buffer.BUFF[477] := 124);
   MBTU_Enable_MBTCP : BOOL := 1;
   MBTU_EnetModulePort : STRING := '$01$00';
   MBTU_Inactivity_Timeout : DINT := 60000;
   MBTU_Log_Enable : DINT := 255;
   MBTU_MB_0xx : BOOL[256] := ([4] := 1, [5] := 1, [96] := 1, [106] := 1, [107] := 1, [111] := 1, [112] := 1, [119] := 1, [124] := 1);
   MBTU_MB_1xx : BOOL[256] := ([1] := 1, [2] := 1, [3] := 1, [4] := 1, [5] := 1, [6] := 1, [17] := 1, [18] := 1);
   MBTU_MB_3xx : INT[1000];
   MBTU_MB_4xx : INT[100] := ([6] := 25, [7] := 24, [8] := 25, [9] := 32, [10] := 125, [11] := 125);
   MBTU_Sock_Accept_Timeout : DINT := 10000;
   RedBypass1 : BOOL;
   RedBypass2 : BOOL;
   RedBypass3 : BOOL;
   RedConnected1 : BOOL;
   RedConnected2 : BOOL;
   RedConnected3 : BOOL;
   RedESTOP1 : ALIAS FOR Red_Driver_Station:I.Data.1;
   RedESTOP1Light : ALIAS FOR Red_Driver_Station:O.Data.15;
   RedESTOP2 : ALIAS FOR Red_Driver_Station:I.Data.3;
   RedESTOP2Light : ALIAS FOR Red_Driver_Station:O.Data.13;
   RedESTOP3 : ALIAS FOR Red_Driver_Station:I.Data.5;
   RedESTOP3Light : ALIAS FOR Red_Driver_Station:O.Data.11;
   RedSoftwareESTOP1 : BOOL;
   RedSoftwareESTOP2 : BOOL;
   RedSoftwareESTOP3 : BOOL;
   RedStackStatus1 : ALIAS FOR Red_Driver_Station:O.Data.14;
   RedStackStatus2 : ALIAS FOR Red_Driver_Station:O.Data.12;
   RedStackStatus3 : ALIAS FOR Red_Driver_Station:O.Data.10;
   Sand_Storm_T1 : TIMER := (PRE := 2000);
   Sand_Storm_T2 : TIMER := (PRE := 2000);
   SL_1 : BOOL;
   SL_2 : BOOL := 1;
   SL_3 : BOOL := 1;
   SL_B : BOOL;
   Stack_Buzzer : ALIAS FOR Local:1:O.Data.5;
   Stack_Buzzer_Timer : TIMER := (PRE := 950);
   Stack_Light_Blue : ALIAS FOR Local:1:O.Data.1;
   Stack_Light_Green : ALIAS FOR Local:1:O.Data.4;
   Stack_Light_Orange : ALIAS FOR Local:1:O.Data.3;
   Stack_Light_Red : ALIAS FOR Local:1:O.Data.2;
   Watchdog : BOOL;
END_VAR

PROGRAM MainProgram   (* main routine JSR *)

ROUTINE Alliance_Stack_Lights   (* ladder *)
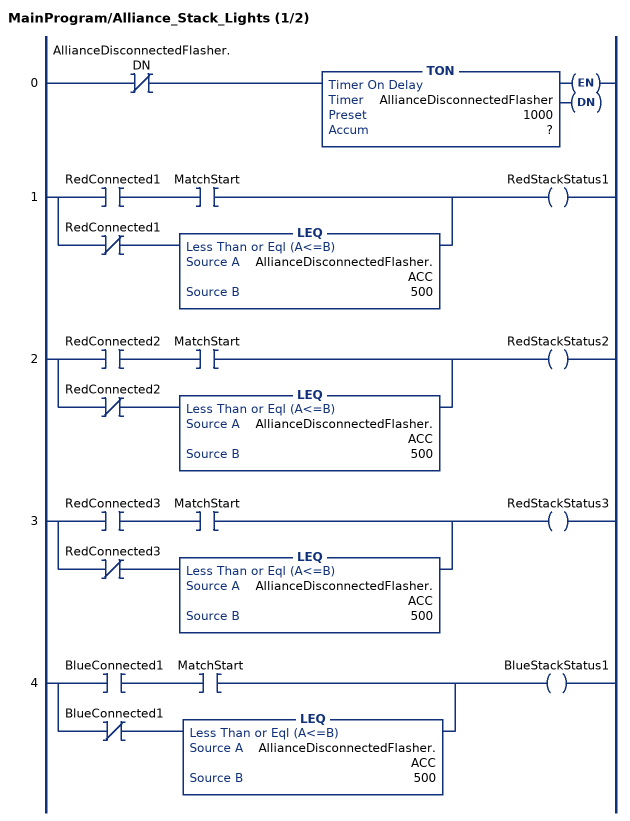
   0: XIO(AllianceDisconnectedFlasher.DN)TON(AllianceDisconnectedFlasher,?,?);
   1: [XIC(RedConnected1) XIC(MatchStart) ,XIO(RedConnected1) LEQ(AllianceDisconnectedFlasher.ACC,500) ]OTE(RedStackStatus1);
   2: [XIC(RedConnected2) XIC(MatchStart) ,XIO(RedConnected2) LEQ(AllianceDisconnectedFlasher.ACC,500) ]OTE(RedStackStatus2);
   3: [XIC(RedConnected3) XIC(MatchStart) ,XIO(RedConnected3) LEQ(AllianceDisconnectedFlasher.ACC,500) ]OTE(RedStackStatus3);
   4: [XIC(BlueConnected1) XIC(MatchStart) ,XIO(BlueConnected1) LEQ(AllianceDisconnectedFlasher.ACC,500) ]OTE(BlueStackStatus1);
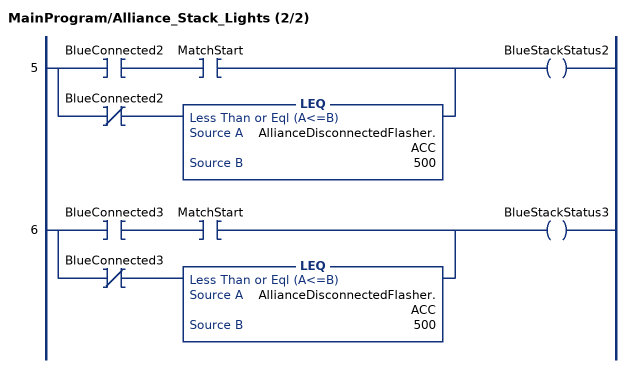
   5: [XIC(BlueConnected2) XIC(MatchStart) ,XIO(BlueConnected2) LEQ(AllianceDisconnectedFlasher.ACC,500) ]OTE(BlueStackStatus2);
   6: [XIC(BlueConnected3) XIC(MatchStart) ,XIO(BlueConnected3) LEQ(AllianceDisconnectedFlasher.ACC,500) ]OTE(BlueStackStatus3);
END_ROUTINE

ROUTINE ESTOP   (* ladder *)
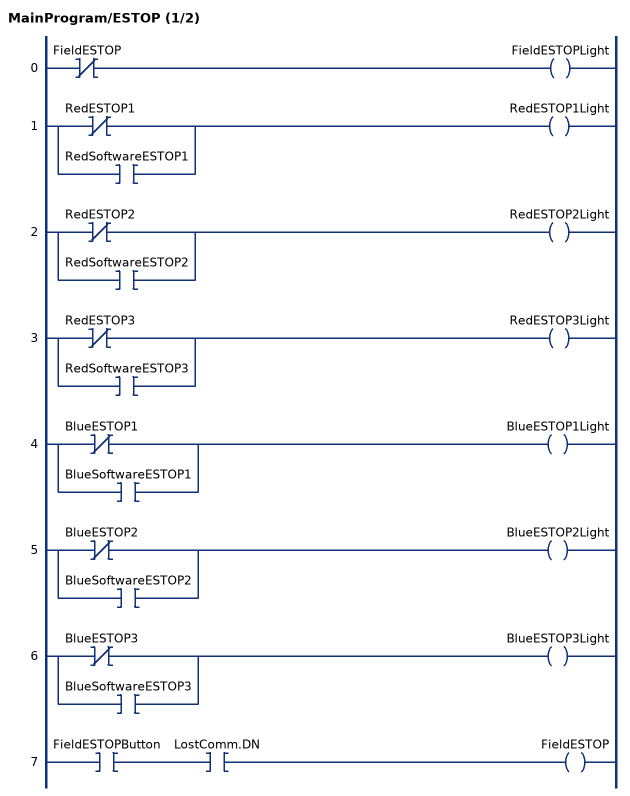
   0: XIO(FieldESTOP)OTE(FieldESTOPLight);
   1: [XIO(RedESTOP1) ,XIC(RedSoftwareESTOP1) ]OTE(RedESTOP1Light);
   2: [XIO(RedESTOP2) ,XIC(RedSoftwareESTOP2) ]OTE(RedESTOP2Light);
   3: [XIO(RedESTOP3) ,XIC(RedSoftwareESTOP3) ]OTE(RedESTOP3Light);
   4: [XIO(BlueESTOP1) ,XIC(BlueSoftwareESTOP1) ]OTE(BlueESTOP1Light);
   5: [XIO(BlueESTOP2) ,XIC(BlueSoftwareESTOP2) ]OTE(BlueESTOP2Light);
   6: [XIO(BlueESTOP3) ,XIC(BlueSoftwareESTOP3) ]OTE(BlueESTOP3Light);
   7: XIC(FieldESTOPButton)XIC(LostComm.DN)OTE(FieldESTOP);
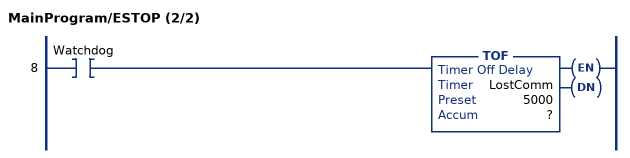
   8: XIC(Watchdog)TOF(LostComm,?,?);
END_ROUTINE

ROUTINE JSR   (* ladder *)
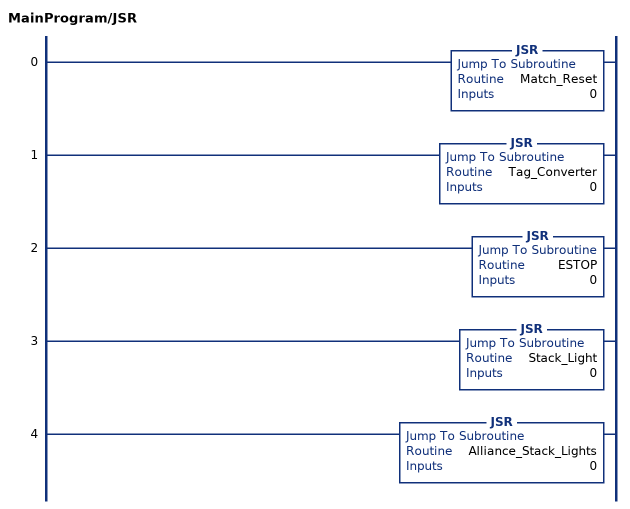
   0: JSR(Match_Reset,0);
   1: JSR(Tag_Converter,0);
   2: JSR(ESTOP,0);
   3: JSR(Stack_Light,0);
   4: JSR(Alliance_Stack_Lights,0);
END_ROUTINE

ROUTINE Match_Reset   (* ladder *)
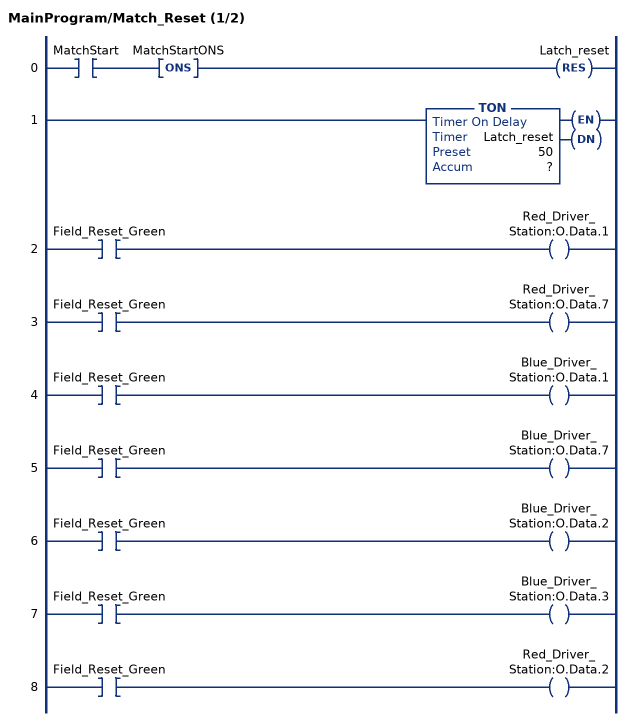
   0: XIC(MatchStart)ONS(MatchStartONS)RES(Latch_reset);
   1: TON(Latch_reset,?,?);
   2: XIC(Field_Reset_Green)OTE(Red_Driver_Station:O.Data.1);
   3: XIC(Field_Reset_Green)OTE(Red_Driver_Station:O.Data.7);
   4: XIC(Field_Reset_Green)OTE(Blue_Driver_Station:O.Data.1);
   5: XIC(Field_Reset_Green)OTE(Blue_Driver_Station:O.Data.7);
   6: XIC(Field_Reset_Green)OTE(Blue_Driver_Station:O.Data.2);
   7: XIC(Field_Reset_Green)OTE(Blue_Driver_Station:O.Data.3);
   8: XIC(Field_Reset_Green)OTE(Red_Driver_Station:O.Data.2);
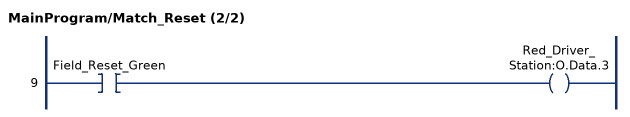
   9: XIC(Field_Reset_Green)OTE(Red_Driver_Station:O.Data.3);
END_ROUTINE

ROUTINE Stack_Light   (* ladder *)
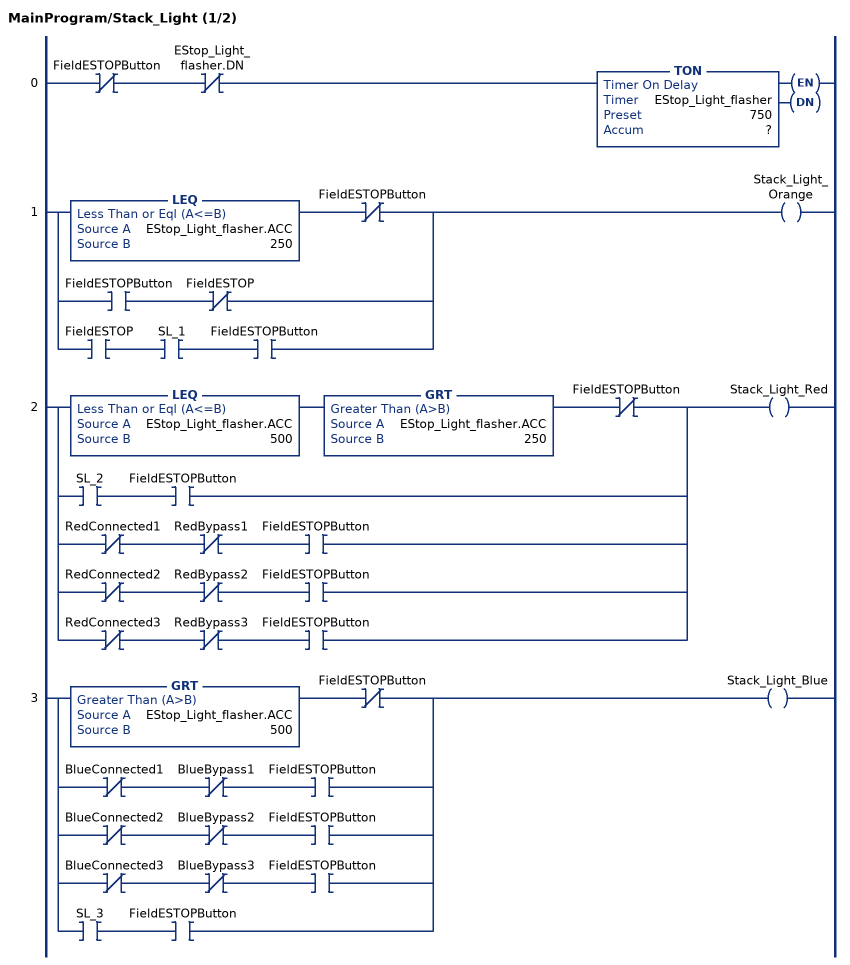
   0: XIO(FieldESTOPButton)XIO(EStop_Light_flasher.DN)TON(EStop_Light_flasher,?,?);
   1: [LEQ(EStop_Light_flasher.ACC,250) XIO(FieldESTOPButton) ,XIC(FieldESTOPButton) XIO(FieldESTOP) ,XIC(FieldESTOP) XIC(SL_1) XIC(FieldESTOPButton) ]OTE(Stack_Light_Orange);
   2: [LEQ(EStop_Light_flasher.ACC,500) GRT(EStop_Light_flasher.ACC,250) XIO(FieldESTOPButton) ,XIC(SL_2) XIC(FieldESTOPButton) ,XIO(RedConnected1) XIO(RedBypass1) XIC(FieldESTOPButton) ,XIO(RedConnected2) XIO(RedBypass2) XIC(FieldESTOPButton) ,XIO(RedConnected3) XIO(RedBypass3) XIC(FieldESTOPButton) ]OTE(Stack_Light_Red);
   3: [GRT(EStop_Light_flasher.ACC,500) XIO(FieldESTOPButton) ,XIO(BlueConnected1) XIO(BlueBypass1) XIC(FieldESTOPButton) ,XIO(BlueConnected2) XIO(BlueBypass2) XIC(FieldESTOPButton) ,XIO(BlueConnected3) XIO(BlueBypass3) XIC(FieldESTOPButton) ,XIC(SL_3) XIC(FieldESTOPButton) ]OTE(Stack_Light_Blue);
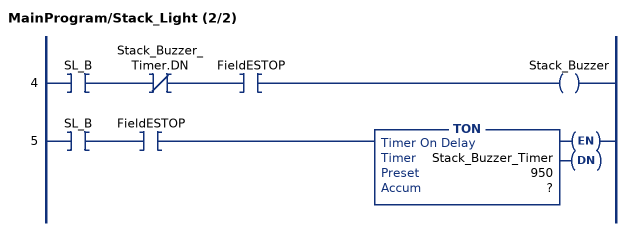
   4: XIC(SL_B)XIO(Stack_Buzzer_Timer.DN)XIC(FieldESTOP)OTE(Stack_Buzzer);
   5: XIC(SL_B)XIC(FieldESTOP)TON(Stack_Buzzer_Timer,?,?);
END_ROUTINE

ROUTINE Tag_Converter   (* ladder *)
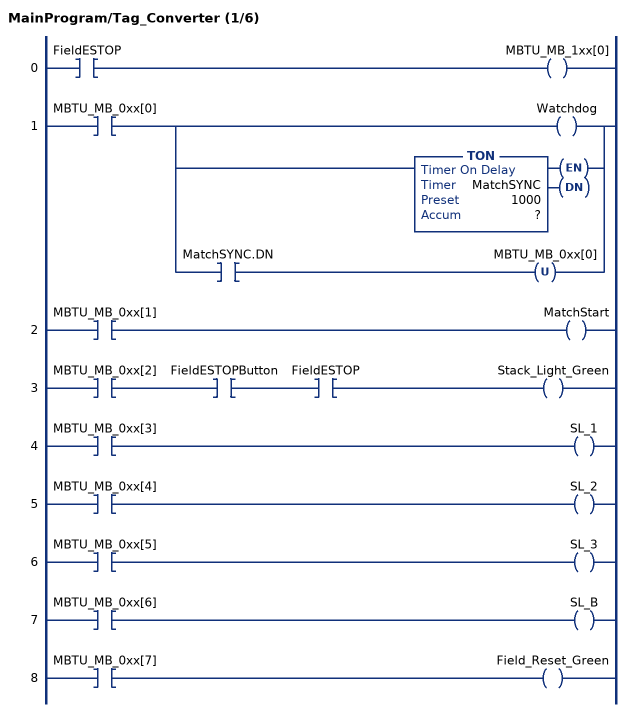
   0: XIC(FieldESTOP)OTE(MBTU_MB_1xx[0]);
   1: XIC(MBTU_MB_0xx[0])[OTE(Watchdog) ,TON(MatchSYNC,?,?) ,XIC(MatchSYNC.DN) OTU(MBTU_MB_0xx[0]) ];
   2: XIC(MBTU_MB_0xx[1])OTE(MatchStart);
   3: XIC(MBTU_MB_0xx[2])XIC(FieldESTOPButton)XIC(FieldESTOP)OTE(Stack_Light_Green);
   4: XIC(MBTU_MB_0xx[3])OTE(SL_1);
   5: XIC(MBTU_MB_0xx[4])OTE(SL_2);
   6: XIC(MBTU_MB_0xx[5])OTE(SL_3);
   7: XIC(MBTU_MB_0xx[6])OTE(SL_B);
   8: XIC(MBTU_MB_0xx[7])OTE(Field_Reset_Green);
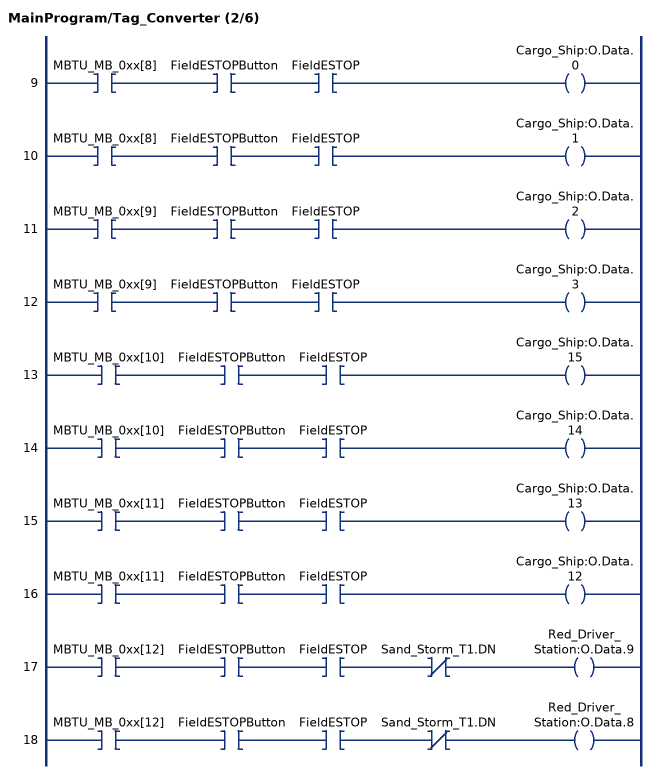
   9: XIC(MBTU_MB_0xx[8])XIC(FieldESTOPButton)XIC(FieldESTOP)OTE(Cargo_Ship:O.Data.0);
   10: XIC(MBTU_MB_0xx[8])XIC(FieldESTOPButton)XIC(FieldESTOP)OTE(Cargo_Ship:O.Data.1);
   11: XIC(MBTU_MB_0xx[9])XIC(FieldESTOPButton)XIC(FieldESTOP)OTE(Cargo_Ship:O.Data.2);
   12: XIC(MBTU_MB_0xx[9])XIC(FieldESTOPButton)XIC(FieldESTOP)OTE(Cargo_Ship:O.Data.3);
   13: XIC(MBTU_MB_0xx[10])XIC(FieldESTOPButton)XIC(FieldESTOP)OTE(Cargo_Ship:O.Data.15);
   14: XIC(MBTU_MB_0xx[10])XIC(FieldESTOPButton)XIC(FieldESTOP)OTE(Cargo_Ship:O.Data.14);
   15: XIC(MBTU_MB_0xx[11])XIC(FieldESTOPButton)XIC(FieldESTOP)OTE(Cargo_Ship:O.Data.13);
   16: XIC(MBTU_MB_0xx[11])XIC(FieldESTOPButton)XIC(FieldESTOP)OTE(Cargo_Ship:O.Data.12);
   17: XIC(MBTU_MB_0xx[12])XIC(FieldESTOPButton)XIC(FieldESTOP)XIO(Sand_Storm_T1.DN)OTE(Red_Driver_Station:O.Data.9);
   18: XIC(MBTU_MB_0xx[12])XIC(FieldESTOPButton)XIC(FieldESTOP)XIO(Sand_Storm_T1.DN)OTE(Red_Driver_Station:O.Data.8);
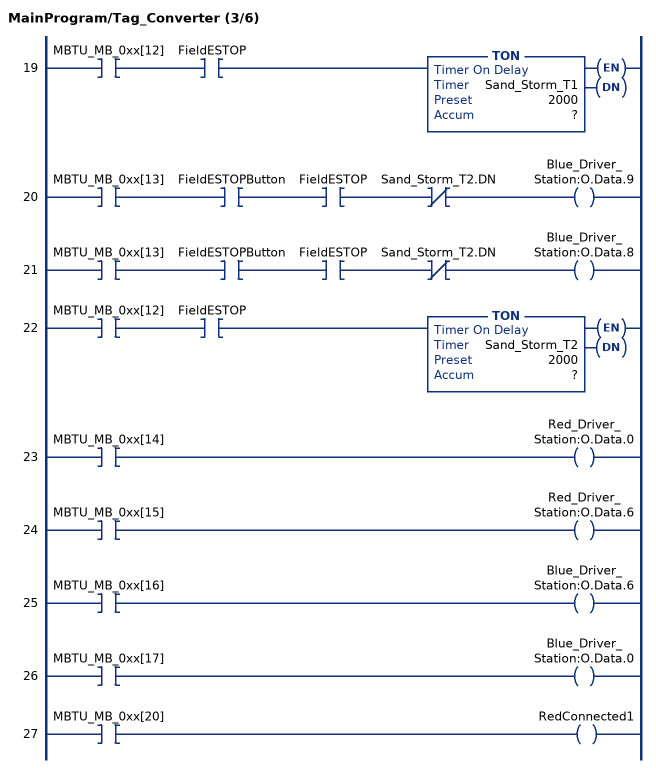
   19: XIC(MBTU_MB_0xx[12])XIC(FieldESTOP)TON(Sand_Storm_T1,?,?);
   20: XIC(MBTU_MB_0xx[13])XIC(FieldESTOPButton)XIC(FieldESTOP)XIO(Sand_Storm_T2.DN)OTE(Blue_Driver_Station:O.Data.9);
   21: XIC(MBTU_MB_0xx[13])XIC(FieldESTOPButton)XIC(FieldESTOP)XIO(Sand_Storm_T2.DN)OTE(Blue_Driver_Station:O.Data.8);
   22: XIC(MBTU_MB_0xx[12])XIC(FieldESTOP)TON(Sand_Storm_T2,?,?);
   23: XIC(MBTU_MB_0xx[14])OTE(Red_Driver_Station:O.Data.0);
   24: XIC(MBTU_MB_0xx[15])OTE(Red_Driver_Station:O.Data.6);
   25: XIC(MBTU_MB_0xx[16])OTE(Blue_Driver_Station:O.Data.6);
   26: XIC(MBTU_MB_0xx[17])OTE(Blue_Driver_Station:O.Data.0);
   27: XIC(MBTU_MB_0xx[20])OTE(RedConnected1);
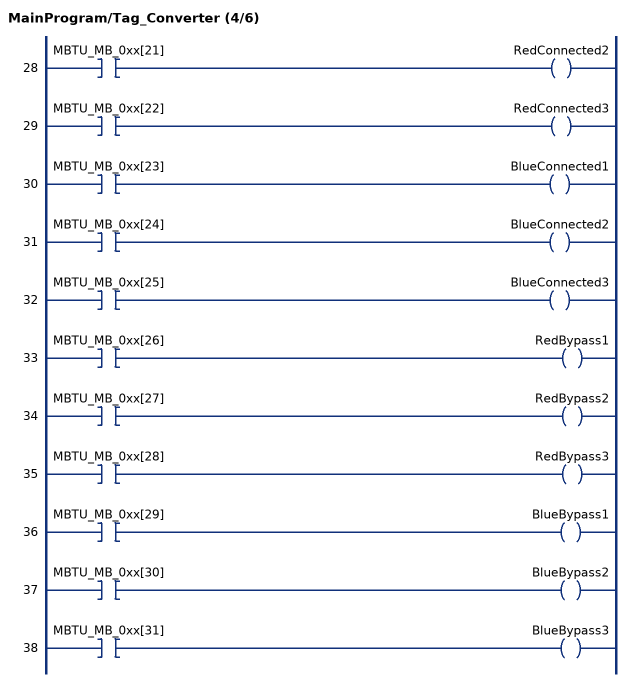
   28: XIC(MBTU_MB_0xx[21])OTE(RedConnected2);
   29: XIC(MBTU_MB_0xx[22])OTE(RedConnected3);
   30: XIC(MBTU_MB_0xx[23])OTE(BlueConnected1);
   31: XIC(MBTU_MB_0xx[24])OTE(BlueConnected2);
   32: XIC(MBTU_MB_0xx[25])OTE(BlueConnected3);
   33: XIC(MBTU_MB_0xx[26])OTE(RedBypass1);
   34: XIC(MBTU_MB_0xx[27])OTE(RedBypass2);
   35: XIC(MBTU_MB_0xx[28])OTE(RedBypass3);
   36: XIC(MBTU_MB_0xx[29])OTE(BlueBypass1);
   37: XIC(MBTU_MB_0xx[30])OTE(BlueBypass2);
   38: XIC(MBTU_MB_0xx[31])OTE(BlueBypass3);
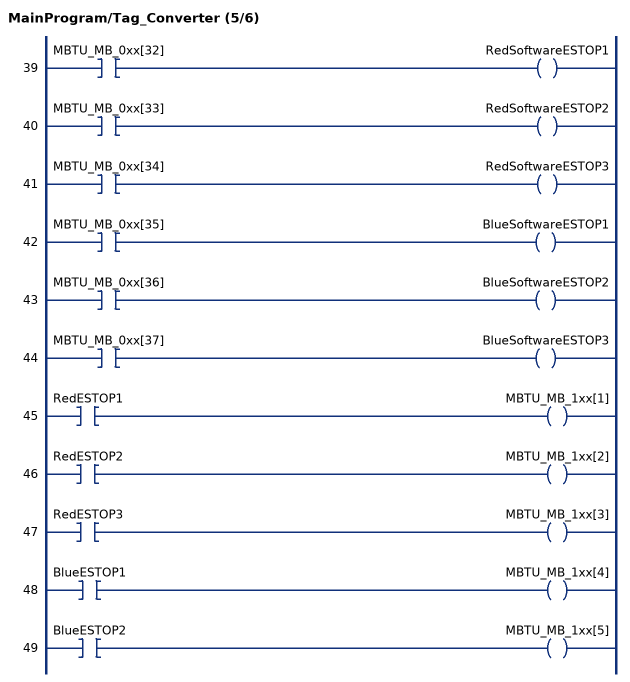
   39: XIC(MBTU_MB_0xx[32])OTE(RedSoftwareESTOP1);
   40: XIC(MBTU_MB_0xx[33])OTE(RedSoftwareESTOP2);
   41: XIC(MBTU_MB_0xx[34])OTE(RedSoftwareESTOP3);
   42: XIC(MBTU_MB_0xx[35])OTE(BlueSoftwareESTOP1);
   43: XIC(MBTU_MB_0xx[36])OTE(BlueSoftwareESTOP2);
   44: XIC(MBTU_MB_0xx[37])OTE(BlueSoftwareESTOP3);
   45: XIC(RedESTOP1)OTE(MBTU_MB_1xx[1]);
   46: XIC(RedESTOP2)OTE(MBTU_MB_1xx[2]);
   47: XIC(RedESTOP3)OTE(MBTU_MB_1xx[3]);
   48: XIC(BlueESTOP1)OTE(MBTU_MB_1xx[4]);
   49: XIC(BlueESTOP2)OTE(MBTU_MB_1xx[5]);
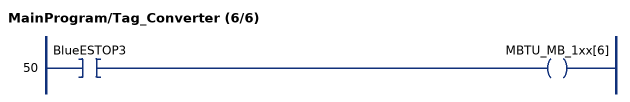
   50: XIC(BlueESTOP3)OTE(MBTU_MB_1xx[6]);
END_ROUTINE
END_PROGRAM

PROGRAM ModbusSlaveTCP   (* main routine Modbus_TCP_Slave *)
VAR
   Additional_len : INT := 6;
   Additional_len_read : INT := 12;
   buff_bit_index : DINT := 5;
   buff_byte_index : DINT := 2;
   CMD_END : DINT := 12;
   CMD_IN : DINT := 2;
   CMD_LEN : DINT := 13;
   CMD_LEN1 : INT := 20;
   CMD_LEN2 : INT := 5;
   CMD_START : DINT;
   Coil_Byte_Count : DINT := 2;
   coil_wr_index : DINT := 2;
   Conn_Open : BOOL[32] := ([10] := 1, [11] := 1, [12] := 1, [13] := 1, [14] := 1, [15] := 1, [16] := 1, [17] := 1, [18] := 1, [19] := 1);
   Data_Received : BOOL;
   EX_CMD : INT := 144;
   EX_CODE : INT := 2;
   Found : BOOL := 1;
   INT_DATA_IN : INT := 1280;
   INT_IN : INT := 2;
   INT_STR_OUT : STRING := '$00$05';
   Listen_Retry_Tmr : TIMER := (PRE := 20);
   Listen_Socket_Lost : BOOL;
   Log_Old : DINT := 255;
   Main_Read_Buffer : STR_4096[20];
   mb_bit_index : DINT := 13;
   MB_Resp_Data : STR_462 := '$02$7F$00';
   MB_TMP_INT : INT := -5632;
   Modbus_Byte_cnt : INT := 240;
   Modbus_Bytes : DINT := 5;
   Modbus_CMD_Len : INT := 3328;
   Modbus_Cmd_String : STR_462 := '$02$00$00$00$0D';
   Modbus_ID : STRING := '$00q$00$00';
   Modbus_Packet : STR_462 := '$00q$00$00$00$06$01$02$00$00$00$0D';
   Modbus_resp_Str : STR_462 := '$00q$00$00$00$05$01$02$02$7F$00';
   Modbus_Ret_CMD : STRING := '$02';
   Modbus_Ret_len : STRING := '$00$05';
   Modbus_Start : INT;
   Modbus_Unit : STRING := '$01';
   Next_Write : BOOL[32];
   No_Open_Sockets : BOOL;
   Nothing : BOOL := 1;
   ONS : BOOL[64] := ([1] := 1, [2] := 1, [3] := 1, [4] := 1, [8] := 1);
   ONS_B : BOOL[32] := ([0] := 1, [1] := 1, [2] := 1, [3] := 1, [4] := 1, [5] := 1, [6] := 1, [7] := 1, [8] := 1, [9] := 1);
   ONS_ERR : BOOL[32] := ([0] := 1, [1] := 1, [2] := 1, [3] := 1, [4] := 1, [5] := 1, [6] := 1, [7] := 1, [8] := 1, [9] := 1, [20] := 1, [21] := 1, [22] := 1, [23] := 1, [24] := 1, [25] := 1, [26] := 1, [27] := 1, [28] := 1, [29] := 1);
   RetryCreateSock : TIMER := (PRE := 2000);
   RG_4x_Pos : DINT := 1;
   RG_STR_TMP : STRING := '$00 ';
   RW_Instance : INT[20];
   RW_Select : DINT := 10;
   Startup_Timer : TIMER := (PRE := 1000, ACC := 1000, EN := 1, DN := 1);
   Str_Out : STR_1 := '$02';
   String_Pos : INT := 246;
   TestCntr : COUNTER := (PRE := 99999, ACC := 4733);
   testint : DINT;
   Valid : BOOL[32];
   Valid_CMD : BOOL[32];
   Valid_Command : BOOL;
   Valid_End : BOOL;
   Valid_Len : BOOL;
   Valid_Len_16 : BOOL;
   Valid_Start_Addr : BOOL;
   Valid_Value_05 : BOOL;
   W_Log_Accept : ALIAS FOR MBTU_Log_Enable.2;
   W_Log_Attribute : ALIAS FOR MBTU_Log_Enable.6;
   W_Log_Create : ALIAS FOR MBTU_Log_Enable.0;
   W_Log_Delete : ALIAS FOR MBTU_Log_Enable.5;
   W_Log_Errors : ALIAS FOR MBTU_Log_Enable.7;
   W_Log_Open : ALIAS FOR MBTU_Log_Enable.1;
   W_Log_Read : ALIAS FOR MBTU_Log_Enable.3;
   W_Log_Write : ALIAS FOR MBTU_Log_Enable.4;
END_VAR

ROUTINE _SUB_0x_RD   (* ladder *)
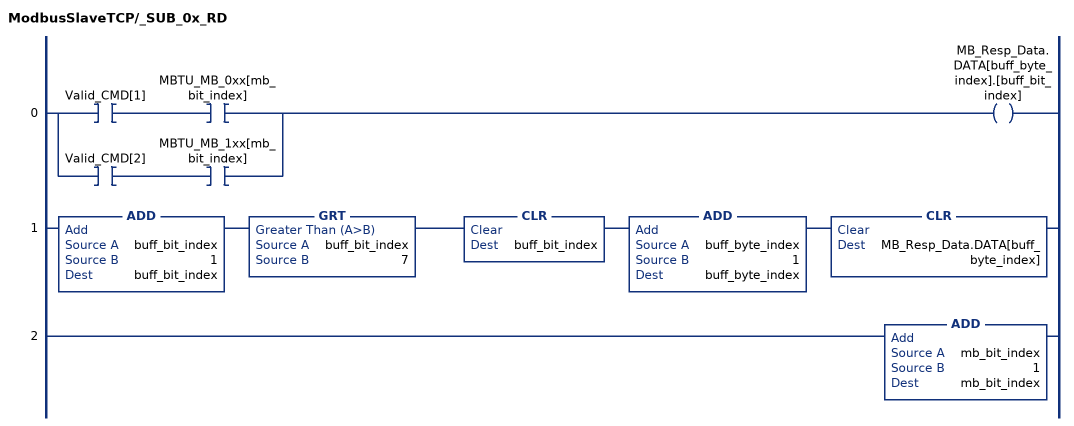
   0: [XIC(Valid_CMD[1]) XIC(MBTU_MB_0xx[mb_bit_index]) ,XIC(Valid_CMD[2]) XIC(MBTU_MB_1xx[mb_bit_index]) ]OTE(MB_Resp_Data.DATA[buff_byte_index].[buff_bit_index]);
   1: ADD(buff_bit_index,1,buff_bit_index)GRT(buff_bit_index,7)CLR(buff_bit_index)ADD(buff_byte_index,1,buff_byte_index)CLR(MB_Resp_Data.DATA[buff_byte_index]);
   2: ADD(mb_bit_index,1,mb_bit_index);
END_ROUTINE

ROUTINE _SUB_0x_WR   (* ladder *)
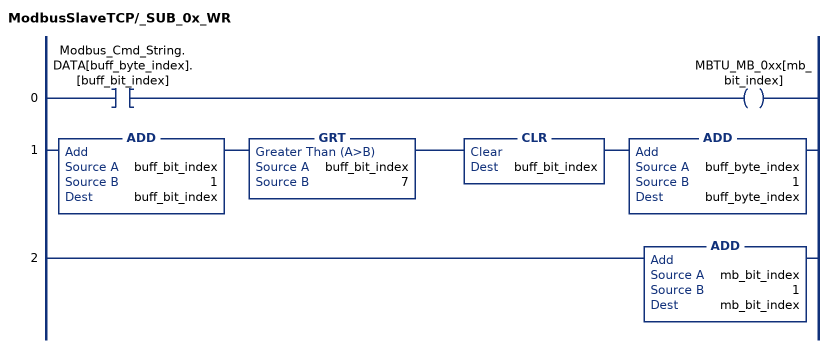
   0: XIC(Modbus_Cmd_String.DATA[buff_byte_index].[buff_bit_index])OTE(MBTU_MB_0xx[mb_bit_index]);
   1: ADD(buff_bit_index,1,buff_bit_index)GRT(buff_bit_index,7)CLR(buff_bit_index)ADD(buff_byte_index,1,buff_byte_index);
   2: ADD(mb_bit_index,1,mb_bit_index);
END_ROUTINE

ROUTINE _SUB_4x_RD   (* ladder *)
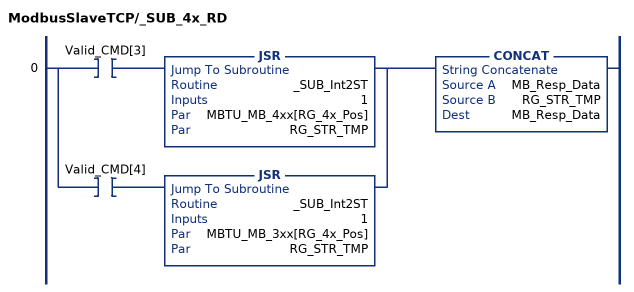
   0: [XIC(Valid_CMD[3]) JSR(_SUB_Int2ST,1,MBTU_MB_4xx[RG_4x_Pos],RG_STR_TMP) ,XIC(Valid_CMD[4]) JSR(_SUB_Int2ST,1,MBTU_MB_3xx[RG_4x_Pos],RG_STR_TMP) ]CONCAT(MB_Resp_Data,RG_STR_TMP,MB_Resp_Data);
END_ROUTINE
